KUKA KRL program: MyProgram_344().src

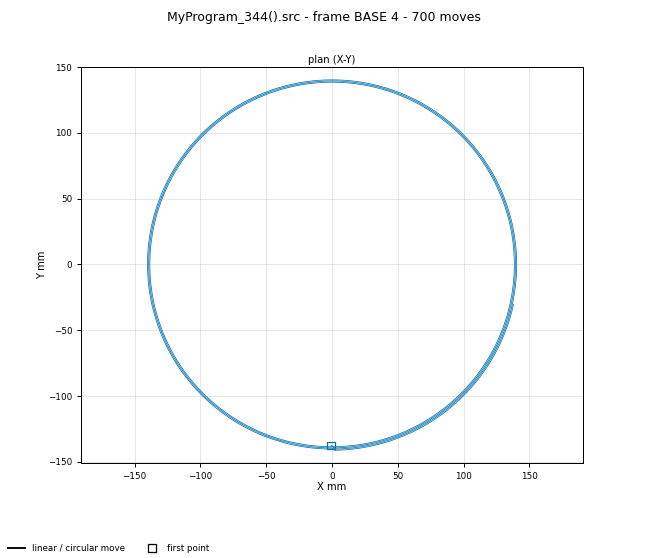
[picture p0: tool path of MyProgram_344().src in frame BASE 4, 700 of 700 moves have a stored position in this frame; points joined in program order, loops and branches not executed]
&ACCESS RVP
&REL 1
&PARAM TEMPLATE = C:\KRC\Roboter\Template\vorgabe
&PARAM EDITMASK = *
DEF MyProgram_344()
; ---- Setting reference (Base) ----
$BASE = BASE_DATA[4]

; --------------------------
; ---- Setting tool (TCP) ----
$TOOL = TOOL_DATA[3]
; --------------------------

$VEL.CP = VEL_APROX_PRINT
Startdeposition()
$VEL.CP = VEL_PRINT
LIN {X -0.555,Y -137.593,Z 192,A -68.2325,B 0.4034,C 0.1604,E1 0.4627,E2 159.7049} C_DIS
Enddeposition()
LIN {X 0.9941,Y -138.4895,Z 192,A -68.6521,B 0.4236,C 0.1629,E1 0.4819,E2 160.302} C_DIS
Startdeposition()
$VEL.CP = VEL_PRINT
LIN {X 0.9941,Y -138.4895,Z 192,A -68.6533,B 0.4236,C 0.1629,E1 0.4819,E2 160.3034} C_DIS
LIN {X -2.5108,Y -138.4702,Z 192,A -70.1889,B 0.423,C 0.1643,E1 0.4773,E2 161.8537} C_DIS
LIN {X -7.0615,Y -138.3127,Z 192,A -71.9031,B 0.4225,C 0.1655,E1 0.4723,E2 163.5419} C_DIS
LIN {X -10.2792,Y -138.1109,Z 192,A -73.1462,B 0.4222,C 0.1664,E1 0.4687,E2 164.7714} C_DIS
LIN {X -14.0249,Y -137.783,Z 192,A -74.535,B 0.4219,C 0.1671,E1 0.4646,E2 166.1344} C_DIS
LIN {X -18.2105,Y -137.2903,Z 192,A -76.1855,B 0.4216,C 0.168,E1 0.4598,E2 167.771} C_DIS
LIN {X -21.5368,Y -136.8082,Z 192,A -77.5051,B 0.4213,C 0.1687,E1 0.4559,E2 169.0801} C_DIS
LIN {X -25.201,Y -136.1828,Z 192,A -78.927,B 0.4211,C 0.1692,E1 0.4518,E2 170.4843} C_DIS
LIN {X -28.0321,Y -135.6266,Z 192,A -80.0916,B 0.4209,C 0.1697,E1 0.4484,E2 171.6448} C_DIS
LIN {X -31.6468,Y -134.8308,Z 192,A -81.5349,B 0.4207,C 0.1701,E1 0.4443,E2 173.0749} C_DIS
LIN {X -34.3072,Y -134.1761,Z 192,A -82.6457,B 0.4206,C 0.1704,E1 0.4411,E2 174.1826} C_DIS
LIN {X -38.108,Y -133.1489,Z 192,A -84.2158,B 0.4205,C 0.1708,E1 0.4366,E2 175.7441} C_DIS
LIN {X -41.3369,Y -132.1821,Z 192,A -85.5836,B 0.4204,C 0.171,E1 0.4327,E2 177.1083} C_DIS
LIN {X -44.1513,Y -131.2668,Z 192,A -86.8094,B 0.4204,C 0.1711,E1 0.4292,E2 178.3348} C_DIS
LIN {X -47.7758,Y -129.9936,Z 192,A -88.3761,B 0.4203,C 0.1711,E1 0.4248,E2 179.8986} C_DIS
LIN {X -50.9793,Y -128.771,Z 192,A -89.8008,B 0.4203,C 0.1711,E1 0.4209,E2 181.325} C_DIS
LIN {X -54.0825,Y -127.4982,Z 192,A -91.2041,B 0.4203,C 0.1711,E1 0.417,E2 182.7313} C_DIS
LIN {X -56.8706,Y -126.2773,Z 192,A -92.5332,B 0.4204,C 0.1709,E1 0.4133,E2 184.0722} C_DIS
LIN {X -60.4865,Y -124.5883,Z 192,A -94.1895,B 0.4206,C 0.1705,E1 0.4089,E2 185.7299} C_DIS
LIN {X -63.61,Y -123.0229,Z 192,A -95.691,B 0.4207,C 0.1701,E1 0.4049,E2 187.2409} C_DIS
LIN {X -66.285,Y -121.6017,Z 192,A -97.0782,B 0.4209,C 0.1697,E1 0.4012,E2 188.65} C_DIS
LIN {X -70.0463,Y -119.4747,Z 192,A -98.9871,B 0.4212,C 0.169,E1 0.3962,E2 190.5788} C_DIS
LIN {X -73.7798,Y -117.2059,Z 192,A -100.9315,B 0.4215,C 0.168,E1 0.3912,E2 192.5456} C_DIS
LIN {X -77.534,Y -114.7569,Z 192,A -102.9321,B 0.422,C 0.1669,E1 0.3862,E2 194.57} C_DIS
LIN {X -81.1785,Y -112.2084,Z 192,A -104.9505,B 0.4225,C 0.1656,E1 0.3813,E2 196.6173} C_DIS
LIN {X -84.7483,Y -109.5372,Z 192,A -106.9996,B 0.4231,C 0.1641,E1 0.3763,E2 198.6993} C_DIS
LIN {X -88.4224,Y -106.5934,Z 192,A -109.1404,B 0.4238,C 0.1623,E1 0.3714,E2 200.871} C_DIS
LIN {X -91.6396,Y -103.8405,Z 192,A -111.1887,B 0.4245,C 0.1605,E1 0.3667,E2 202.9667} C_DIS
LIN {X -94.9496,Y -100.8229,Z 192,A -113.3283,B 0.4253,C 0.1584,E1 0.362,E2 205.1518} C_DIS
LIN {X -98.1617,Y -97.6982,Z 192,A -115.4971,B 0.4261,C 0.156,E1 0.3573,E2 207.3704} C_DIS
LIN {X -101.2932,Y -94.4476,Z 192,A -117.7031,B 0.4271,C 0.1535,E1 0.3527,E2 209.6298} C_DIS
LIN {X -104.4308,Y -90.9664,Z 192,A -119.9695,B 0.4281,C 0.1506,E1 0.3482,E2 211.9476} C_DIS
LIN {X -107.1621,Y -87.7323,Z 192,A -122.1746,B 0.4291,C 0.1477,E1 0.344,E2 214.2236} C_DIS
LIN {X -110.0811,Y -84.0406,Z 192,A -124.5209,B 0.4303,C 0.1443,E1 0.3397,E2 216.6321} C_DIS
LIN {X -112.6171,Y -80.6104,Z 192,A -126.7728,B 0.4314,C 0.1409,E1 0.3357,E2 218.9595} C_DIS
LIN {X -115.2516,Y -76.7967,Z 192,A -129.1574,B 0.4326,C 0.1371,E1 0.3317,E2 221.4161} C_DIS
LIN {X -117.5235,Y -73.2728,Z 192,A -131.4426,B 0.4338,C 0.1333,E1 0.328,E2 223.7857} C_DIS
LIN {X -119.9181,Y -69.2845,Z 192,A -133.8851,B 0.4351,C 0.129,E1 0.3243,E2 226.3071} C_DIS
LIN {X -121.9449,Y -65.6516,Z 192,A -136.1958,B 0.4363,C 0.1248,E1 0.321,E2 228.7072} C_DIS
LIN {X -123.5969,Y -62.4824,Z 192,A -138.0865,B 0.4373,C 0.1211,E1 0.3184,E2 230.6599} C_DIS
LIN {X -125.339,Y -58.9152,Z 192,A -140.2644,B 0.4385,C 0.1168,E1 0.3157,E2 232.9182} C_DIS
LIN {X -126.7762,Y -55.7554,Z 192,A -142.2121,B 0.4395,C 0.1129,E1 0.3133,E2 234.9421} C_DIS
LIN {X -128.1275,Y -52.5756,Z 192,A -144.1677,B 0.4406,C 0.1088,E1 0.3111,E2 236.9756} C_DIS
LIN {X -129.393,Y -49.3792,Z 192,A -146.1301,B 0.4416,C 0.1047,E1 0.309,E2 239.0175} C_DIS
LIN {X -130.5727,Y -46.1694,Z 192,A -148.0979,B 0.4426,C 0.1004,E1 0.307,E2 241.0662} C_DIS
LIN {X -131.4708,Y -43.5386,Z 192,A -149.7078,B 0.4434,C 0.0968,E1 0.3055,E2 242.7429} C_DIS
LIN {X -132.529,Y -40.2034,Z 192,A -151.7407,B 0.4443,C 0.0922,E1 0.3037,E2 244.8603} C_DIS
LIN {X -133.4355,Y -37.0832,Z 192,A -153.656,B 0.4452,C 0.0878,E1 0.3022,E2 246.8574} C_DIS
LIN {X -134.2916,Y -33.8522,Z 192,A -155.631,B 0.4461,C 0.0832,E1 0.3007,E2 248.9165} C_DIS
LIN {X -135.1229,Y -30.3677,Z 192,A -157.7323,B 0.447,C 0.0782,E1 0.2993,E2 251.1051} C_DIS
LIN {X -135.8753,Y -26.8097,Z 192,A -159.9357,B 0.4479,C 0.0729,E1 0.298,E2 253.4062} C_DIS
LIN {X -136.6401,Y -22.5773,Z 192,A -162.5203,B 0.4489,C 0.0665,E1 0.2967,E2 256.102} C_DIS
LIN {X -137.1281,Y -19.3939,Z 192,A -164.4714,B 0.4496,C 0.0617,E1 0.2959,E2 258.1376} C_DIS
LIN {X -137.6124,Y -15.6101,Z 192,A -166.7803,B 0.4504,C 0.0559,E1 0.2951,E2 260.5455} C_DIS
LIN {X -138.0192,Y -11.4448,Z 192,A -169.4132,B 0.4511,C 0.0493,E1 0.2943,E2 263.2988} C_DIS
LIN {X -138.3076,Y -7.1633,Z 192,A -172.0124,B 0.4518,C 0.0427,E1 0.2939,E2 266.0064} C_DIS
LIN {X -138.4451,Y -3.6396,Z 192,A -174.1874,B 0.4523,C 0.0371,E1 0.2937,E2 268.2745} C_DIS
LIN {X -138.4943,Y -0.3953,Z 192,A -176.1959,B 0.4527,C 0.0319,E1 0.2937,E2 270.3685} C_DIS
LIN {X -138.4702,Y 2.5108,Z 192,A -177.963,B 0.453,C 0.0274,E1 0.2937,E2 272.2073} C_DIS
LIN {X -138.3076,Y 7.1633,Z 192,A 179.1755,B 0.4534,C 0.02,E1 0.2941,E2 275.1859} C_DIS
LIN {X -138.3076,Y 7.1633,Z 192,A 179.1746,B 0.4534,C 0.02,E1 0.2941,E2 275.1869} C_DIS
LIN {X -137.9693,Y 12.0354,Z 192,A 176.2175,B 0.4536,C 0.0124,E1 0.2947,E2 278.2592} C_DIS
LIN {X -137.9693,Y 12.0354,Z 192,A 176.2165,B 0.4536,C 0.0124,E1 0.2947,E2 278.2602} C_DIS
LIN {X -137.6124,Y 15.6101,Z 192,A 174.0658,B 0.4538,C 0.0069,E1 0.2954,E2 280.4913} C_DIS
LIN {X -137.214,Y 18.7931,Z 192,A 172.1065,B 0.4538,C 0.0019,E1 0.2961,E2 282.5262} C_DIS
LIN {X -136.7379,Y 21.9909,Z 192,A 170.138,B 0.4538,C -0.0031,E1 0.297,E2 284.569} C_DIS
LIN {X -136.2264,Y 24.9574,Z 192,A 168.3314,B 0.4538,C -0.0076,E1 0.2979,E2 286.4408} C_DIS
LIN {X -135.5475,Y 28.4205,Z 192,A 166.1798,B 0.4536,C -0.013,E1 0.2991,E2 288.6719} C_DIS
LIN {X -134.8308,Y 31.6468,Z 192,A 164.192,B 0.4535,C -0.0179,E1 0.3004,E2 290.7298} C_DIS
LIN {X -134.0315,Y 34.877,Z 192,A 162.2011,B 0.4532,C -0.0227,E1 0.3018,E2 292.7892} C_DIS
LIN {X -133.2966,Y 37.5799,Z 192,A 160.5251,B 0.453,C -0.0267,E1 0.3031,E2 294.522} C_DIS
LIN {X -132.1821,Y 41.3369,Z 192,A 158.2172,B 0.4527,C -0.0322,E1 0.3051,E2 296.9044} C_DIS
LIN {X -131.1305,Y 44.5606,Z 192,A 156.2264,B 0.4523,C -0.0368,E1 0.3069,E2 298.9579} C_DIS
LIN {X -130.0987,Y 47.4843,Z 192,A 154.4441,B 0.452,C -0.0409,E1 0.3087,E2 300.7927} C_DIS
LIN {X -128.9199,Y 50.5962,Z 192,A 152.4488,B 0.4515,C -0.0453,E1 0.3108,E2 302.8522} C_DIS
LIN {X -127.4626,Y 54.1678,Z 192,A 150.2777,B 0.451,C -0.0501,E1 0.3132,E2 305.082} C_DIS
LIN {X -126.0683,Y 57.338,Z 192,A 148.3077,B 0.4505,C -0.0543,E1 0.3156,E2 307.106} C_DIS
LIN {X -124.5883,Y 60.4865,Z 192,A 146.3461,B 0.45,C -0.0584,E1 0.3181,E2 309.1192} C_DIS
LIN {X -123.0229,Y 63.61,Z 192,A 144.3948,B 0.4495,C -0.0624,E1 0.3207,E2 311.1199} C_DIS
LIN {X -121.5263,Y 66.4232,Z 192,A 142.5706,B 0.449,C -0.066,E1 0.3232,E2 312.9928} C_DIS
LIN {X -119.4747,Y 70.0463,Z 192,A 140.2278,B 0.4483,C -0.0704,E1 0.3267,E2 315.3943} C_DIS
LIN {X -117.1798,Y 73.8211,Z 192,A 137.8387,B 0.4476,C -0.0748,E1 0.3304,E2 317.8354} C_DIS
LIN {X -114.7569,Y 77.534,Z 192,A 135.4725,B 0.4469,C -0.0789,E1 0.3343,E2 320.2501} C_DIS
LIN {X -112.2084,Y 81.1785,Z 192,A 133.1307,B 0.4462,C -0.0828,E1 0.3383,E2 322.6369} C_DIS
LIN {X -109.5372,Y 84.7483,Z 192,A 130.8146,B 0.4455,C -0.0865,E1 0.3424,E2 324.9946} C_DIS
LIN {X -106.5934,Y 88.4224,Z 192,A 128.4626,B 0.4448,C -0.09,E1 0.3468,E2 327.3815} C_DIS
LIN {X -103.8405,Y 91.6396,Z 192,A 126.265,B 0.4442,C -0.0931,E1 0.3511,E2 329.6173} C_DIS
LIN {X -100.8229,Y 94.9496,Z 192,A 124.0464,B 0.4435,C -0.096,E1 0.3556,E2 331.8666} C_DIS
LIN {X -97.6982,Y 98.1617,Z 192,A 121.8322,B 0.4429,C -0.0987,E1 0.3603,E2 334.1107} C_DIS
LIN {X -94.2952,Y 101.4351,Z 192,A 119.6016,B 0.4424,C -0.1012,E1 0.3651,E2 336.3638} C_DIS
LIN {X -90.9664,Y 104.4308,Z 192,A 117.4631,B 0.4419,C -0.1034,E1 0.3699,E2 338.5252} C_DIS
LIN {X -87.7323,Y 107.1621,Z 192,A 115.4142,B 0.4414,C -0.1053,E1 0.3746,E2 340.598} C_DIS
LIN {X -84.0406,Y 110.0811,Z 192,A 113.2812,B 0.441,C -0.1072,E1 0.3796,E2 342.7453} C_DIS
LIN {X -80.4554,Y 112.728,Z 192,A 111.2383,B 0.4406,C -0.1087,E1 0.3845,E2 344.8035} C_DIS
LIN {X -76.9626,Y 115.1409,Z 192,A 109.2749,B 0.4403,C -0.11,E1 0.3894,E2 346.783} C_DIS
LIN {X -73.2728,Y 117.5235,Z 192,A 107.304,B 0.44,C -0.1111,E1 0.3944,E2 348.7653} C_DIS
LIN {X -69.2845,Y 119.9181,Z 192,A 105.3033,B 0.4397,C -0.1121,E1 0.3995,E2 350.7712} C_DIS
LIN {X -65.7176,Y 121.9094,Z 192,A 103.4573,B 0.4396,C -0.1128,E1 0.4044,E2 352.629} C_DIS
LIN {X -62.0516,Y 123.8162,Z 192,A 101.7909,B 0.4394,C -0.1134,E1 0.4088,E2 354.2911} C_DIS
LIN {X -59.3101,Y 125.1503,Z 192,A 100.4556,B 0.4394,C -0.1137,E1 0.4124,E2 355.6316} C_DIS
LIN {X -55.7554,Y 126.7762,Z 192,A 98.838,B 0.4393,C -0.114,E1 0.4168,E2 357.2487} C_DIS
LIN {X -52.5756,Y 128.1275,Z 192,A 97.3919,B 0.4393,C -0.1141,E1 0.4208,E2 358.6955} C_DIS
LIN {X -49.6556,Y 129.2856,Z 192,A 96.0714,B 0.4393,C -0.1141,E1 0.4245,E2 360.017} C_DIS
LIN {X -46.1694,Y 130.5727,Z 192,A 94.5588,B 0.4393,C -0.1141,E1 0.4287,E2 361.527} C_DIS
LIN {X -42.9496,Y 131.667,Z 192,A 93.172,B 0.4393,C -0.114,E1 0.4326,E2 362.9116} C_DIS
LIN {X -39.967,Y 132.6014,Z 192,A 91.8954,B 0.4393,C -0.1137,E1 0.4362,E2 364.1863} C_DIS
LIN {X -36.4926,Y 133.6007,Z 192,A 90.4567,B 0.4394,C -0.1134,E1 0.4404,E2 365.6199} C_DIS
LIN {X -33.2616,Y 134.4415,Z 192,A 89.1274,B 0.4395,C -0.1131,E1 0.4442,E2 366.9444} C_DIS
LIN {X -30.033,Y 135.1994,Z 192,A 87.817,B 0.4396,C -0.1126,E1 0.448,E2 368.2492} C_DIS
LIN {X -27.3611,Y 135.7631,Z 192,A 86.6941,B 0.4397,C -0.1121,E1 0.4513,E2 369.3711} C_DIS
LIN {X -23.5946,Y 136.4703,Z 192,A 85.2526,B 0.4399,C -0.1115,E1 0.4554,E2 370.8004} C_DIS
LIN {X -20.3903,Y 136.9857,Z 192,A 83.9977,B 0.4401,C -0.1108,E1 0.4591,E2 372.0478} C_DIS
LIN {X -17.1996,Y 137.4228,Z 192,A 82.7606,B 0.4402,C -0.1101,E1 0.4627,E2 373.2766} C_DIS
LIN {X -13.0223,Y 137.8793,Z 192,A 81.1595,B 0.4405,C -0.1091,E1 0.4674,E2 374.8657} C_DIS
LIN {X -9.967,Y 138.1337,Z 192,A 79.9863,B 0.4407,C -0.1083,E1 0.4709,E2 376.0306} C_DIS
LIN {X -6.1741,Y 138.3573,Z 192,A 78.5706,B 0.441,C -0.1072,E1 0.475,E2 377.4331} C_DIS
LIN {X -3.6396,Y 138.4451,Z 192,A 77.5718,B 0.4412,C -0.1063,E1 0.478,E2 378.4273} C_DIS
LIN {X 0,Y 138.495,Z 192,A 76.2697,B 0.4414,C -0.1053,E1 0.4818,E2 379.712} C_DIS
LIN {X 4.1288,Y 138.4315,Z 192,A 74.7561,B 0.4418,C -0.1039,E1 0.4862,E2 381.2087} C_DIS
LIN {X 7.1633,Y 138.3076,Z 192,A 73.5697,B 0.442,C -0.1027,E1 0.4897,E2 382.3889} C_DIS
LIN {X 10.8687,Y 138.0678,Z 192,A 72.2626,B 0.4423,C -0.1014,E1 0.4935,E2 383.6763} C_DIS
LIN {X 14.0249,Y 137.783,Z 192,A 71.1092,B 0.4426,C -0.1001,E1 0.4968,E2 384.8159} C_DIS
LIN {X 18.3405,Y 137.2733,Z 192,A 69.5037,B 0.443,C -0.0983,E1 0.5015,E2 386.4043} C_DIS
LIN {X 21.9321,Y 136.747,Z 192,A 68.2316,B 0.4434,C -0.0968,E1 0.5051,E2 387.6564} C_DIS
LIN {X 24.721,Y 136.2687,Z 192,A 67.1837,B 0.4436,C -0.0955,E1 0.5081,E2 388.6932} C_DIS
LIN {X 28.4205,Y 135.5475,Z 192,A 65.879,B 0.444,C -0.0939,E1 0.5118,E2 389.9755} C_DIS
LIN {X 32.7749,Y 134.5588,Z 192,A 64.2612,B 0.4445,C -0.0917,E1 0.5164,E2 391.5725} C_DIS
LIN {X 36.4926,Y 133.6007,Z 192,A 62.9482,B 0.4448,C -0.0899,E1 0.52,E2 392.8609} C_DIS
LIN {X 39.7229,Y 132.6761,Z 192,A 61.7715,B 0.4451,C -0.0882,E1 0.5233,E2 394.0183} C_DIS
LIN {X 42.5024,Y 131.8098,Z 192,A 60.724,B 0.4455,C -0.0867,E1 0.5261,E2 395.0513} C_DIS
LIN {X 46.1694,Y 130.5727,Z 192,A 59.4127,B 0.4458,C -0.0847,E1 0.5297,E2 396.3362} C_DIS
LIN {X 49.3792,Y 129.393,Z 192,A 58.2311,B 0.4462,C -0.0829,E1 0.5328,E2 397.4964} C_DIS
LIN {X 52.0629,Y 128.3342,Z 192,A 57.2312,B 0.4465,C -0.0813,E1 0.5355,E2 398.4782} C_DIS
LIN {X 55.7554,Y 126.7762,Z 192,A 55.8629,B 0.4469,C -0.0791,E1 0.5391,E2 399.8196} C_DIS
LIN {X 58.4713,Y 125.5442,Z 192,A 54.811,B 0.4472,C -0.0773,E1 0.5418,E2 400.8542} C_DIS
LIN {X 62.7685,Y 123.4512,Z 192,A 53.2475,B 0.4476,C -0.0747,E1 0.5458,E2 402.3785} C_DIS
LIN {X 65.9341,Y 121.7931,Z 192,A 51.9114,B 0.448,C -0.0723,E1 0.5491,E2 403.7011} C_DIS
LIN {X 69.7683,Y 119.638,Z 192,A 50.4277,B 0.4484,C -0.0696,E1 0.5528,E2 405.1525} C_DIS
LIN {X 73.5368,Y 117.3592,Z 192,A 48.9472,B 0.4488,C -0.0669,E1 0.5563,E2 406.6} C_DIS
LIN {X 77.2651,Y 114.939,Z 192,A 47.4954,B 0.4492,C -0.0643,E1 0.5597,E2 408.0139} C_DIS
LIN {X 80.9148,Y 112.3995,Z 192,A 46.0136,B 0.4496,C -0.0615,E1 0.5631,E2 409.4604} C_DIS
LIN {X 84.4903,Y 109.7372,Z 192,A 44.4994,B 0.45,C -0.0585,E1 0.5665,E2 410.9417} C_DIS
LIN {X 87.9854,Y 106.9552,Z 192,A 43.0481,B 0.4504,C -0.0556,E1 0.5696,E2 412.3531} C_DIS
LIN {X 91.3943,Y 104.0574,Z 192,A 41.5465,B 0.4508,C -0.0526,E1 0.5728,E2 413.8193} C_DIS
LIN {X 94.7112,Y 101.0477,Z 192,A 40.0745,B 0.4511,C -0.0496,E1 0.5758,E2 415.2523} C_DIS
LIN {X 97.9307,Y 97.9307,Z 192,A 38.6398,B 0.4514,C -0.0467,E1 0.5786,E2 416.6436} C_DIS
LIN {X 101.0477,Y 94.7112,Z 192,A 37.1759,B 0.4517,C -0.0436,E1 0.5814,E2 418.0669} C_DIS
LIN {X 103.9957,Y 91.4641,Z 192,A 35.739,B 0.452,C -0.0405,E1 0.5841,E2 419.464} C_DIS
LIN {X 106.9552,Y 87.9854,Z 192,A 34.2626,B 0.4523,C -0.0374,E1 0.5867,E2 420.8964} C_DIS
LIN {X 109.7372,Y 84.4903,Z 192,A 32.8039,B 0.4525,C -0.0342,E1 0.5891,E2 422.3133} C_DIS
LIN {X 112.3995,Y 80.9148,Z 192,A 31.3402,B 0.4528,C -0.0309,E1 0.5915,E2 423.7358} C_DIS
LIN {X 114.939,Y 77.2651,Z 192,A 29.9377,B 0.453,C -0.0279,E1 0.5937,E2 425.0905} C_DIS
LIN {X 117.352,Y 73.5484,Z 192,A 28.5103,B 0.4531,C -0.0247,E1 0.5958,E2 426.4731} C_DIS
LIN {X 119.638,Y 69.7683,Z 192,A 27.0552,B 0.4533,C -0.0213,E1 0.5978,E2 427.8868} C_DIS
LIN {X 121.875,Y 65.7816,Z 192,A 25.6074,B 0.4535,C -0.0181,E1 0.5997,E2 429.2848} C_DIS
LIN {X 123.8162,Y 62.0516,Z 192,A 24.332,B 0.4535,C -0.0152,E1 0.6013,E2 430.5074} C_DIS
LIN {X 125.339,Y 58.9152,Z 192,A 23.2157,B 0.4536,C -0.0127,E1 0.6026,E2 431.5864} C_DIS
LIN {X 126.7762,Y 55.7554,Z 192,A 22.1058,B 0.4536,C -0.0101,E1 0.6038,E2 432.6588} C_DIS
LIN {X 127.9883,Y 52.9089,Z 192,A 21.1185,B 0.4537,C -0.0078,E1 0.6049,E2 433.6121} C_DIS
LIN {X 129.393,Y 49.3792,Z 192,A 19.9048,B 0.4537,C -0.005,E1 0.6061,E2 434.784} C_DIS
LIN {X 130.361,Y 46.7567,Z 192,A 19.0109,B 0.4538,C -0.0029,E1 0.6069,E2 435.647} C_DIS
LIN {X 131.5332,Y 43.3512,Z 192,A 17.8438,B 0.4538,C -0.0001,E1 0.6079,E2 436.776} C_DIS
LIN {X 132.6761,Y 39.7229,Z 192,A 16.6541,B 0.4538,C 0.0026,E1 0.6088,E2 437.92} C_DIS
LIN {X 133.8705,Y 35.4808,Z 192,A 15.2396,B 0.4538,C 0.006,E1 0.6098,E2 439.2855} C_DIS
LIN {X 134.8308,Y 31.6468,Z 192,A 13.9948,B 0.4538,C 0.0089,E1 0.6106,E2 440.4832} C_DIS
LIN {X 135.5475,Y 28.4205,Z 192,A 12.9443,B 0.4537,C 0.0114,E1 0.6112,E2 441.4951} C_DIS
LIN {X 136.1828,Y 25.201,Z 192,A 11.9014,B 0.4536,C 0.0139,E1 0.6118,E2 442.4996} C_DIS
LIN {X 136.8951,Y 20.9756,Z 192,A 10.5272,B 0.4535,C 0.0172,E1 0.6124,E2 443.8247} C_DIS
LIN {X 137.4228,Y 17.1996,Z 192,A 9.3297,B 0.4534,C 0.02,E1 0.6128,E2 444.9751} C_DIS
LIN {X 137.8793,Y 13.0223,Z 192,A 7.9962,B 0.4532,C 0.0232,E1 0.6132,E2 446.258} C_DIS
LIN {X 138.1406,Y 9.8725,Z 192,A 6.9929,B 0.4531,C 0.0256,E1 0.6134,E2 447.223} C_DIS
LIN {X 138.3357,Y 6.6024,Z 192,A 5.959,B 0.4529,C 0.028,E1 0.6135,E2 448.2163} C_DIS
LIN {X 138.4451,Y 3.6396,Z 192,A 4.9707,B 0.4528,C 0.0304,E1 0.6136,E2 449.1745} C_DIS
LIN {X 138.4943,Y 0.3953,Z 192,A 3.9518,B 0.4526,C 0.0328,E1 0.6136,E2 450.1521} C_DIS
LIN {X 138.4608,Y -3.074,Z 192,A 2.875,B 0.4524,C 0.0353,E1 0.6136,E2 451.1829} C_DIS
LIN {X 138.3076,Y -7.1633,Z 192,A 1.5785,B 0.4522,C 0.0384,E1 0.6134,E2 452.4282} C_DIS
LIN {X 138.087,Y -10.6067,Z 192,A 0.4731,B 0.452,C 0.041,E1 0.6132,E2 453.4917} C_DIS
LIN {X 137.783,Y -14.0249,Z 192,A -0.625,B 0.4517,C 0.0436,E1 0.6129,E2 454.548} C_DIS
LIN {X 137.4921,Y -16.6185,Z 192,A -1.5008,B 0.4515,C 0.0458,E1 0.6127,E2 455.3971} C_DIS
LIN {X 136.9857,Y -20.3903,Z 192,A -2.673,B 0.4512,C 0.0484,E1 0.6122,E2 456.5163} C_DIS
LIN {X 136.4839,Y -23.5132,Z 192,A -3.6749,B 0.451,C 0.0508,E1 0.6118,E2 457.4775} C_DIS
LIN {X 135.8753,Y -26.8097,Z 192,A -4.7551,B 0.4507,C 0.0533,E1 0.6113,E2 458.517} C_DIS
LIN {X 135.1994,Y -30.033,Z 192,A -5.8083,B 0.4504,C 0.0558,E1 0.6107,E2 459.5289} C_DIS
LIN {X 134.4416,Y -33.2616,Z 192,A -6.8713,B 0.4501,C 0.0582,E1 0.61,E2 460.5505} C_DIS
LIN {X 133.7106,Y -36.0806,Z 192,A -7.826,B 0.4498,C 0.0605,E1 0.6093,E2 461.4714} C_DIS
LIN {X 132.6761,Y -39.7229,Z 192,A -9.016,B 0.4494,C 0.0632,E1 0.6084,E2 462.6105} C_DIS
LIN {X 131.667,Y -42.9496,Z 192,A -10.1007,B 0.449,C 0.0656,E1 0.6075,E2 463.6524} C_DIS
LIN {X 130.5727,Y -46.1694,Z 192,A -11.1926,B 0.4487,C 0.0681,E1 0.6066,E2 464.7013} C_DIS
LIN {X 129.59,Y -48.8533,Z 192,A -12.1224,B 0.4483,C 0.0702,E1 0.6057,E2 465.5964} C_DIS
LIN {X 128.1275,Y -52.5756,Z 192,A -13.3979,B 0.4479,C 0.0731,E1 0.6044,E2 466.8197} C_DIS
LIN {X 126.7762,Y -55.7554,Z 192,A -14.5111,B 0.4475,C 0.0756,E1 0.6032,E2 467.8892} C_DIS
LIN {X 125.339,Y -58.9152,Z 192,A -15.6306,B 0.447,C 0.0781,E1 0.602,E2 468.9647} C_DIS
LIN {X 123.8968,Y -61.8883,Z 192,A -16.693,B 0.4466,C 0.0804,E1 0.6007,E2 469.9845} C_DIS
LIN {X 122.3814,Y -64.8316,Z 192,A -17.7503,B 0.4462,C 0.0827,E1 0.5994,E2 470.9981} C_DIS
LIN {X 120.5157,Y -68.2408,Z 192,A -19.0826,B 0.4456,C 0.0857,E1 0.5976,E2 472.2919} C_DIS
LIN {X 118.2823,Y -72.0428,Z 192,A -20.5134,B 0.445,C 0.0888,E1 0.5956,E2 473.6671} C_DIS
LIN {X 115.9812,Y -75.691,Z 192,A -21.9254,B 0.4444,C 0.0918,E1 0.5936,E2 475.0263} C_DIS
LIN {X 113.4302,Y -79.4635,Z 192,A -23.3998,B 0.4438,C 0.0949,E1 0.5913,E2 476.4424} C_DIS
LIN {X 110.8167,Y -83.0694,Z 192,A -24.8543,B 0.4431,C 0.0979,E1 0.5889,E2 477.8414} C_DIS
LIN {X 108.101,Y -86.5737,Z 192,A -26.327,B 0.4424,C 0.1009,E1 0.5865,E2 479.2621} C_DIS
LIN {X 105.2302,Y -90.0415,Z 192,A -27.7831,B 0.4418,C 0.1038,E1 0.5839,E2 480.6596} C_DIS
LIN {X 102.2647,Y -93.3958,Z 192,A -29.2565,B 0.4411,C 0.1067,E1 0.5812,E2 482.078} C_DIS
LIN {X 99.2163,Y -96.6279,Z 192,A -30.7254,B 0.4404,C 0.1096,E1 0.5784,E2 483.4932} C_DIS
LIN {X 96.011,Y -99.8135,Z 192,A -32.2504,B 0.4396,C 0.1126,E1 0.5754,E2 484.9679} C_DIS
LIN {X 92.7324,Y -102.8667,Z 192,A -33.7377,B 0.4389,C 0.1154,E1 0.5724,E2 486.4016} C_DIS
LIN {X 89.5033,Y -105.6877,Z 192,A -35.0973,B 0.4383,C 0.1178,E1 0.5696,E2 487.6999} C_DIS
LIN {X 86.1302,Y -108.454,Z 192,A -36.5622,B 0.4375,C 0.1205,E1 0.5664,E2 489.1147} C_DIS
LIN {X 82.6157,Y -111.1545,Z 192,A -38.052,B 0.4368,C 0.1231,E1 0.5632,E2 490.5535} C_DIS
LIN {X 79.0004,Y -113.7524,Z 192,A -39.5497,B 0.436,C 0.1258,E1 0.5598,E2 492.0001} C_DIS
LIN {X 75.5139,Y -116.0962,Z 192,A -41.0032,B 0.4353,C 0.1283,E1 0.5564,E2 493.4114} C_DIS
LIN {X 71.7664,Y -118.4494,Z 192,A -42.5021,B 0.4346,C 0.1308,E1 0.5528,E2 494.8607} C_DIS
LIN {X 67.9604,Y -120.6733,Z 192,A -44.0032,B 0.4338,C 0.1332,E1 0.5492,E2 496.3135} C_DIS
LIN {X 64.0989,Y -122.7662,Z 192,A -45.4473,B 0.4331,C 0.1354,E1 0.5457,E2 497.7011} C_DIS
LIN {X 60.4865,Y -124.5883,Z 192,A -46.8242,B 0.4325,C 0.1375,E1 0.5422,E2 499.0334} C_DIS
LIN {X 57.7806,Y -125.8636,Z 192,A -47.8847,B 0.4319,C 0.1392,E1 0.5395,E2 500.0672} C_DIS
LIN {X 54.1678,Y -127.4626,Z 192,A -49.2201,B 0.4313,C 0.1411,E1 0.536,E2 501.3574} C_DIS
LIN {X 50.9793,Y -128.771,Z 192,A -50.4163,B 0.4308,C 0.1428,E1 0.5329,E2 502.5188} C_DIS
LIN {X 48.0728,Y -129.8823,Z 192,A -51.5145,B 0.4302,C 0.1444,E1 0.53,E2 503.5883} C_DIS
LIN {X 44.5606,Y -131.1305,Z 192,A -52.8035,B 0.4297,C 0.1461,E1 0.5266,E2 504.8388} C_DIS
LIN {X 41.9266,Y -131.9938,Z 192,A -53.7841,B 0.4292,C 0.1474,E1 0.5239,E2 505.7942} C_DIS
LIN {X 38.6732,Y -132.9834,Z 192,A -54.9796,B 0.4287,C 0.1489,E1 0.5207,E2 506.9575} C_DIS
LIN {X 34.877,Y -134.0315,Z 192,A -56.3689,B 0.4281,C 0.1507,E1 0.5168,E2 508.3102} C_DIS
LIN {X 31.6468,Y -134.8308,Z 192,A -57.5522,B 0.4276,C 0.1521,E1 0.5135,E2 509.4641} C_DIS
LIN {X 28.4205,Y -135.5475,Z 192,A -58.7326,B 0.4271,C 0.1535,E1 0.5102,E2 510.6159} C_DIS
LIN {X 25.201,Y -136.1828,Z 192,A -59.9103,B 0.4266,C 0.1548,E1 0.5069,E2 511.7661} C_DIS
LIN {X 22.4273,Y -136.6651,Z 192,A -60.953,B 0.4262,C 0.156,E1 0.504,E2 512.7903} C_DIS
LIN {X 18.7931,Y -137.214,Z 192,A -62.2549,B 0.4257,C 0.1573,E1 0.5003,E2 514.0586} C_DIS
LIN {X 15.6101,Y -137.6124,Z 192,A -63.4217,B 0.4252,C 0.1585,E1 0.4969,E2 515.2009} C_DIS
LIN {X 11.4448,Y -138.0192,Z 192,A -64.9524,B 0.4247,C 0.1599,E1 0.4925,E2 516.7008} C_DIS
LIN {X 8.3309,Y -138.2421,Z 192,A -66.1418,B 0.4243,C 0.1611,E1 0.4891,E2 517.8748} C_DIS
LIN {X 4.6209,Y -138.4179,Z 192,A -67.4751,B 0.4239,C 0.1621,E1 0.4852,E2 519.1767} C_DIS
LIN {X 1.5336,Y -138.4865,Z 192,A -68.6233,B 0.4235,C 0.1631,E1 0.4819,E2 520.3051} C_DIS
LIN {X 1.5336,Y -138.4865,Z 192,A -68.6233,B 0.4235,C 0.1631,E1 0.4819,E2 520.3051} C_DIS
Enddeposition()
LIN {X 1.0026,Y -139.3847,Z 192,A -69.1006,B 0.4435,C 0.1645,E1 0.5006,E2 520.8324} C_DIS
Startdeposition()
$VEL.CP = VEL_PRINT
LIN {X 4.2647,Y -139.327,Z 192,A -67.6877,B 0.444,C 0.1631,E1 0.5048,E2 519.4071} C_DIS
LIN {X 8.4179,Y -139.1373,Z 192,A -66.1532,B 0.4445,C 0.1618,E1 0.5092,E2 517.8995} C_DIS
LIN {X 12.2098,Y -138.8567,Z 192,A -64.8025,B 0.4449,C 0.1606,E1 0.5131,E2 516.5817} C_DIS
LIN {X 15.533,Y -138.5248,Z 192,A -63.5851,B 0.4453,C 0.1595,E1 0.5166,E2 515.3884} C_DIS
LIN {X 18.4825,Y -138.1613,Z 192,A -62.4978,B 0.4457,C 0.1584,E1 0.5197,E2 514.3216} C_DIS
LIN {X 22.1548,Y -137.6219,Z 192,A -61.0215,B 0.4463,C 0.1566,E1 0.5239,E2 512.8521} C_DIS
LIN {X 29.1089,Y -136.3185,Z 192,A -58.742,B 0.447,C 0.1546,E1 0.5302,E2 510.671} C_DIS
LIN {X 33.2706,Y -135.364,Z 192,A -57.0664,B 0.4478,C 0.1523,E1 0.5349,E2 509.0067} C_DIS
LIN {X 35.8565,Y -134.7007,Z 192,A -56.0558,B 0.4482,C 0.151,E1 0.5378,E2 508.009} C_DIS
LIN {X 39.3465,Y -133.723,Z 192,A -54.798,B 0.4488,C 0.1495,E1 0.5412,E2 506.7871} C_DIS
LIN {X 43.33,Y -132.4877,Z 192,A -53.3837,B 0.4493,C 0.1477,E1 0.545,E2 505.4191} C_DIS
LIN {X 45.9063,Y -131.6154,Z 192,A -52.3661,B 0.4498,C 0.1462,E1 0.5477,E2 504.4164} C_DIS
LIN {X 49.3442,Y -130.366,Z 192,A -51.1206,B 0.4504,C 0.1446,E1 0.551,E2 503.2106} C_DIS
LIN {X 52.5632,Y -129.1017,Z 192,A -49.8788,B 0.4509,C 0.1428,E1 0.5543,E2 501.996} C_DIS
LIN {X 56.147,Y -127.5857,Z 192,A -48.2348,B 0.4519,C 0.1398,E1 0.5587,E2 500.3437} C_DIS
LIN {X 59.6467,Y -125.9857,Z 192,A -47.3378,B 0.452,C 0.1393,E1 0.5607,E2 499.5532} C_DIS
LIN {X 62.4051,Y -124.6442,Z 192,A -46.1726,B 0.4526,C 0.1373,E1 0.5637,E2 498.402} C_DIS
LIN {X 65.3981,Y -123.0993,Z 192,A -45.016,B 0.4532,C 0.1355,E1 0.5666,E2 497.28} C_DIS
LIN {X 69.6684,Y -120.7345,Z 192,A -43.2878,B 0.454,C 0.1326,E1 0.5708,E2 495.5937} C_DIS
LIN {X 73.349,Y -118.5348,Z 192,A -41.8003,B 0.4548,C 0.1301,E1 0.5744,E2 494.1476} C_DIS
LIN {X 77.1511,Y -116.0959,Z 192,A -40.2722,B 0.4555,C 0.1275,E1 0.5779,E2 492.669} C_DIS
LIN {X 80.8132,Y -113.5773,Z 192,A -38.7551,B 0.4562,C 0.1249,E1 0.5814,E2 491.1984} C_DIS
LIN {X 84.4876,Y -110.8709,Z 192,A -37.2394,B 0.4569,C 0.1222,E1 0.5847,E2 489.7368} C_DIS
LIN {X 87.9766,Y -108.1234,Z 192,A -35.7468,B 0.4576,C 0.1195,E1 0.5879,E2 488.294} C_DIS
LIN {X 91.3702,Y -105.2714,Z 192,A -34.2501,B 0.4584,C 0.1168,E1 0.5911,E2 486.8457} C_DIS
LIN {X 94.8453,Y -102.1512,Z 192,A -32.7127,B 0.4591,C 0.1139,E1 0.5942,E2 485.3652} C_DIS
LIN {X 98.0714,Y -99.0582,Z 192,A -31.2421,B 0.4598,C 0.1111,E1 0.5971,E2 483.9488} C_DIS
LIN {X 101.1735,Y -95.8878,Z 192,A -29.7481,B 0.4605,C 0.1082,E1 0.5999,E2 482.5033} C_DIS
LIN {X 104.2757,Y -92.5046,Z 192,A -28.2613,B 0.4611,C 0.1053,E1 0.6026,E2 481.0754} C_DIS
LIN {X 107.1472,Y -89.163,Z 192,A -26.7883,B 0.4618,C 0.1023,E1 0.6052,E2 479.6518} C_DIS
LIN {X 109.995,Y -85.625,Z 192,A -25.3246,B 0.4624,C 0.0994,E1 0.6077,E2 478.247} C_DIS
LIN {X 112.5674,Y -82.2142,Z 192,A -23.9253,B 0.4631,C 0.0965,E1 0.61,E2 476.8995} C_DIS
LIN {X 115.0601,Y -78.6872,Z 192,A -22.5102,B 0.4637,C 0.0935,E1 0.6122,E2 475.5364} C_DIS
LIN {X 117.6047,Y -74.8315,Z 192,A -20.6367,B 0.4646,C 0.0888,E1 0.615,E2 473.6653} C_DIS
LIN {X 120.1464,Y -70.6775,Z 192,A -19.6955,B 0.4647,C 0.0881,E1 0.6162,E2 472.8786} C_DIS
LIN {X 120.1464,Y -70.6775,Z 192,A -19.6964,B 0.4647,C 0.0881,E1 0.6162,E2 472.8797} C_DIS
LIN {X 122.5672,Y -66.3921,Z 192,A -17.7973,B 0.4656,C 0.0834,E1 0.6187,E2 470.9972} C_DIS
LIN {X 124.383,Y -62.9196,Z 192,A -16.6332,B 0.466,C 0.0811,E1 0.6201,E2 469.8967} C_DIS
LIN {X 126.5614,Y -58.4133,Z 192,A -14.9731,B 0.4666,C 0.0773,E1 0.6221,E2 468.2926} C_DIS
LIN {X 128.3062,Y -54.4805,Z 192,A -13.6205,B 0.4671,C 0.0744,E1 0.6235,E2 466.9986} C_DIS
LIN {X 129.3571,Y -51.9297,Z 192,A -12.7257,B 0.4674,C 0.0724,E1 0.6244,E2 466.1372} C_DIS
LIN {X 130.6249,Y -48.6532,Z 192,A -11.5589,B 0.4678,C 0.0697,E1 0.6256,E2 465.0088} C_DIS
LIN {X 132.0167,Y -44.7445,Z 192,A -10.287,B 0.4682,C 0.0669,E1 0.6267,E2 463.7974} C_DIS
LIN {X 133.4569,Y -40.2433,Z 192,A -8.6937,B 0.4688,C 0.0631,E1 0.628,E2 462.252} C_DIS
LIN {X 134.6136,Y -36.1831,Z 192,A -7.2259,B 0.4692,C 0.0595,E1 0.629,E2 460.8206} C_DIS
LIN {X 135.5807,Y -32.3716,Z 192,A -5.8428,B 0.4697,C 0.0561,E1 0.6299,E2 459.4691} C_DIS
LIN {X 136.4371,Y -28.5567,Z 192,A -4.8899,B 0.4699,C 0.0545,E1 0.6304,E2 458.6062} C_DIS
LIN {X 137.3359,Y -23.8607,Z 192,A -3.2127,B 0.4703,C 0.0503,E1 0.6312,E2 456.9675} C_DIS
LIN {X 138.0134,Y -19.5534,Z 192,A -1.9435,B 0.4706,C 0.0475,E1 0.6317,E2 455.7689} C_DIS
LIN {X 138.4308,Y -16.3389,Z 192,A -0.8806,B 0.4709,C 0.045,E1 0.6321,E2 454.7418} C_DIS
LIN {X 138.8778,Y -11.9596,Z 192,A 0.5088,B 0.4712,C 0.0417,E1 0.6324,E2 453.4083} C_DIS
LIN {X 139.141,Y -8.3588,Z 192,A 1.655,B 0.4714,C 0.039,E1 0.6326,E2 452.3067} C_DIS
LIN {X 139.3276,Y -4.2436,Z 192,A 3.006,B 0.4716,C 0.0358,E1 0.6328,E2 451.0006} C_DIS
LIN {X 139.3947,Y -0.1243,Z 192,A 4.4075,B 0.4719,C 0.0323,E1 0.6328,E2 449.6371} C_DIS
LIN {X 139.3394,Y 3.8203,Z 192,A 5.5738,B 0.4721,C 0.0297,E1 0.6328,E2 448.53} C_DIS
LIN {X 139.1528,Y 8.1669,Z 192,A 7.0007,B 0.4723,C 0.0262,E1 0.6325,E2 447.1496} C_DIS
LIN {X 138.8567,Y 12.2098,Z 192,A 8.1984,B 0.4724,C 0.0236,E1 0.6323,E2 446.0122} C_DIS
LIN {X 138.5248,Y 15.533,Z 192,A 9.2595,B 0.4725,C 0.021,E1 0.632,E2 444.9908} C_DIS
LIN {X 138.1379,Y 18.6612,Z 192,A 10.3814,B 0.4726,C 0.0182,E1 0.6316,E2 443.8907} C_DIS
LIN {X 136.9262,Y 26.0997,Z 192,A 12.4898,B 0.4728,C 0.0137,E1 0.6307,E2 441.907} C_DIS
LIN {X 136.2976,Y 29.206,Z 192,A 13.7567,B 0.4728,C 0.0102,E1 0.63,E2 440.644} C_DIS
LIN {X 135.4313,Y 32.9914,Z 192,A 14.9795,B 0.4729,C 0.0074,E1 0.6292,E2 439.4675} C_DIS
LIN {X 134.1535,Y 37.8534,Z 192,A 16.5766,B 0.4729,C 0.0036,E1 0.6281,E2 437.9281} C_DIS
LIN {X 133.2162,Y 41.0297,Z 192,A 17.6079,B 0.4729,C 0.0013,E1 0.6273,E2 436.937} C_DIS
LIN {X 132.1757,Y 44.2671,Z 192,A 18.7183,B 0.4729,C -0.0014,E1 0.6263,E2 435.8615} C_DIS
LIN {X 130.9939,Y 47.6515,Z 192,A 19.8955,B 0.4729,C -0.0042,E1 0.6253,E2 434.7199} C_DIS
LIN {X 129.7206,Y 51.0174,Z 192,A 21.0148,B 0.4729,C -0.0067,E1 0.6242,E2 433.6439} C_DIS
LIN {X 128.4502,Y 54.1356,Z 192,A 22.0812,B 0.4729,C -0.0092,E1 0.6231,E2 432.6152} C_DIS
LIN {X 126.3456,Y 58.8801,Z 192,A 23.7028,B 0.4729,C -0.0128,E1 0.6213,E2 431.054} C_DIS
LIN {X 124.6065,Y 62.4807,Z 192,A 25.0421,B 0.4727,C -0.016,E1 0.6197,E2 429.7504} C_DIS
LIN {X 123.3792,Y 64.865,Z 192,A 25.8712,B 0.4727,C -0.0178,E1 0.6186,E2 428.9529} C_DIS
LIN {X 121.3906,Y 68.5189,Z 192,A 27.2894,B 0.4725,C -0.0212,E1 0.6167,E2 427.5685} C_DIS
LIN {X 119.1608,Y 72.3272,Z 192,A 28.747,B 0.4724,C -0.0245,E1 0.6147,E2 426.1518} C_DIS
LIN {X 116.7074,Y 76.2233,Z 192,A 30.22,B 0.4722,C -0.0278,E1 0.6125,E2 424.7267} C_DIS
LIN {X 114.189,Y 79.9469,Z 192,A 31.6878,B 0.472,C -0.031,E1 0.6102,E2 423.3018} C_DIS
LIN {X 111.5491,Y 83.5908,Z 192,A 33.1554,B 0.4718,C -0.0342,E1 0.6078,E2 421.8769} C_DIS
LIN {X 106.2142,Y 90.2718,Z 192,A 35.77,B 0.4713,C -0.0396,E1 0.6034,E2 419.3619} C_DIS
LIN {X 103.8016,Y 93.036,Z 192,A 37.1247,B 0.4711,C -0.0427,E1 0.6009,E2 418.0239} C_DIS
LIN {X 100.8057,Y 96.2739,Z 192,A 38.5942,B 0.4708,C -0.0458,E1 0.5981,E2 416.5917} C_DIS
LIN {X 97.4969,Y 99.6235,Z 192,A 40.879,B 0.4702,C -0.0515,E1 0.5933,E2 414.2688} C_DIS
LIN {X 92.0941,Y 104.6385,Z 192,A 42.5812,B 0.4699,C -0.0539,E1 0.59,E2 412.7094} C_DIS
LIN {X 88.4825,Y 107.7099,Z 192,A 44.1709,B 0.4695,C -0.0571,E1 0.5866,E2 411.1575} C_DIS
LIN {X 84.9257,Y 110.5358,Z 192,A 45.6273,B 0.4692,C -0.0598,E1 0.5834,E2 409.7439} C_DIS
LIN {X 81.4228,Y 113.1413,Z 192,A 47.1327,B 0.4688,C -0.0627,E1 0.58,E2 408.2684} C_DIS
LIN {X 77.6359,Y 115.7722,Z 192,A 48.6673,B 0.4684,C -0.0656,E1 0.5765,E2 406.7708} C_DIS
LIN {X 73.9057,Y 118.1884,Z 192,A 50.1473,B 0.4681,C -0.0682,E1 0.573,E2 405.3261} C_DIS
LIN {X 70.1493,Y 120.4561,Z 192,A 51.6538,B 0.4676,C -0.0709,E1 0.5693,E2 403.8495} C_DIS
LIN {X 66.2279,Y 122.6557,Z 192,A 53.1326,B 0.4673,C -0.0734,E1 0.5657,E2 402.4076} C_DIS
LIN {X 63.2269,Y 124.2266,Z 192,A 54.5666,B 0.4668,C -0.0762,E1 0.562,E2 400.9695} C_DIS
LIN {X 59.6253,Y 125.996,Z 192,A 55.3015,B 0.4668,C -0.0766,E1 0.5603,E2 400.3243} C_DIS
LIN {X 56.7138,Y 127.3322,Z 192,A 56.7047,B 0.4663,C -0.0793,E1 0.5566,E2 398.913} C_DIS
LIN {X 53.4714,Y 128.7276,Z 192,A 57.9109,B 0.466,C -0.0812,E1 0.5534,E2 397.7305} C_DIS
LIN {X 50.4214,Y 129.9523,Z 192,A 59.1029,B 0.4656,C -0.0831,E1 0.5502,E2 396.5541} C_DIS
LIN {X 46.0995,Y 131.5484,Z 192,A 60.7168,B 0.4652,C -0.0855,E1 0.5459,E2 394.9671} C_DIS
LIN {X 42.5746,Y 132.7304,Z 192,A 61.9407,B 0.4649,C -0.0872,E1 0.5426,E2 393.7722} C_DIS
LIN {X 36.9926,Y 134.3943,Z 192,A 63.9757,B 0.4643,C -0.09,E1 0.537,E2 391.7713} C_DIS
LIN {X 33.2993,Y 135.3571,Z 192,A 65.4211,B 0.464,C -0.0921,E1 0.533,E2 390.3377} C_DIS
LIN {X 26.5335,Y 136.8433,Z 192,A 67.64,B 0.4634,C -0.0946,E1 0.5268,E2 388.177} C_DIS
LIN {X 22.0285,Y 137.6417,Z 192,A 69.3897,B 0.463,C -0.0968,E1 0.5218,E2 386.4398} C_DIS
LIN {X 19.4541,Y 138.0276,Z 192,A 70.3788,B 0.4627,C -0.098,E1 0.5189,E2 385.4582} C_DIS
LIN {X 15.2916,Y 138.5508,Z 192,A 71.9344,B 0.4624,C -0.0997,E1 0.5144,E2 383.9183} C_DIS
LIN {X 11.6141,Y 138.907,Z 192,A 73.2631,B 0.4621,C -0.101,E1 0.5106,E2 382.6069} C_DIS
LIN {X 7.9984,Y 139.1632,Z 192,A 74.5422,B 0.4618,C -0.1022,E1 0.5069,E2 381.3471} C_DIS
LIN {X 4.356,Y 139.3245,Z 192,A 75.9841,B 0.4615,C -0.1037,E1 0.5027,E2 379.9107} C_DIS
LIN {X 0.1943,Y 139.3928,Z 192,A 77.4224,B 0.4612,C -0.1048,E1 0.4985,E2 378.4968} C_DIS
LIN {X -3.2616,Y 139.3549,Z 192,A 78.8778,B 0.4609,C -0.1061,E1 0.4942,E2 377.0389} C_DIS
LIN {X -7.2181,Y 139.2049,Z 192,A 80.2469,B 0.4607,C -0.107,E1 0.4902,E2 375.6928} C_DIS
LIN {X -11.2598,Y 138.9369,Z 192,A 81.8572,B 0.4605,C -0.1081,E1 0.4855,E2 374.0878} C_DIS
LIN {X -18.0822,Y 138.2138,Z 192,A 84.4669,B 0.4601,C -0.1096,E1 0.4779,E2 371.4974} C_DIS
LIN {X -26.4375,Y 136.8617,Z 192,A 88.2365,B 0.4596,C -0.1116,E1 0.4668,E2 367.7043} C_DIS
LIN {X -30.9741,Y 135.9065,Z 192,A 89.2498,B 0.4597,C -0.1114,E1 0.4641,E2 366.7678} C_DIS
LIN {X -30.9741,Y 135.9065,Z 192,A 89.2489,B 0.4597,C -0.1114,E1 0.4641,E2 366.7688} C_DIS
LIN {X -34.5652,Y 135.0381,Z 192,A 90.9466,B 0.4595,C -0.112,E1 0.4592,E2 365.0567} C_DIS
LIN {X -37.7202,Y 134.1908,Z 192,A 92.3328,B 0.4595,C -0.1123,E1 0.4552,E2 363.6675} C_DIS
LIN {X -41.031,Y 133.2158,Z 192,A 93.6999,B 0.4595,C -0.1125,E1 0.4513,E2 362.3053} C_DIS
LIN {X -44.4967,Y 132.0992,Z 192,A 95.2051,B 0.4594,C -0.1126,E1 0.4471,E2 360.8001} C_DIS
LIN {X -47.6758,Y 130.9852,Z 192,A 96.5481,B 0.4594,C -0.1126,E1 0.4434,E2 359.4611} C_DIS
LIN {X -50.4971,Y 129.9229,Z 192,A 97.8626,B 0.4594,C -0.1126,E1 0.4397,E2 358.1409} C_DIS
LIN {X -56.3622,Y 127.4895,Z 192,A 100.3909,B 0.4595,C -0.1121,E1 0.4328,E2 355.6207} C_DIS
LIN {X -59.0492,Y 126.2674,Z 192,A 101.9048,B 0.4595,C -0.1119,E1 0.4287,E2 354.0819} C_DIS
LIN {X -62.3429,Y 124.6749,Z 192,A 103.2992,B 0.4597,C -0.1114,E1 0.425,E2 352.6976} C_DIS
LIN {X -65.5693,Y 123.0094,Z 192,A 105.0107,B 0.4598,C -0.1108,E1 0.4204,E2 350.9682} C_DIS
LIN {X -70.7316,Y 120.1146,Z 192,A 108.4111,B 0.4601,C -0.1096,E1 0.4115,E2 347.4849} C_DIS
LIN {X -76.1706,Y 116.7416,Z 192,A 110.319,B 0.4605,C -0.1078,E1 0.4069,E2 345.6413} C_DIS
LIN {X -82.2843,Y 112.5159,Z 192,A 113.4759,B 0.4611,C -0.1054,E1 0.3993,E2 342.4773} C_DIS
LIN {X -84.6675,Y 110.7334,Z 192,A 115.1249,B 0.4614,C -0.1042,E1 0.3953,E2 340.7918} C_DIS
LIN {X -88.2213,Y 107.9234,Z 192,A 117.2528,B 0.4618,C -0.1022,E1 0.3904,E2 338.6414} C_DIS
LIN {X -91.8496,Y 104.8532,Z 192,A 119.4841,B 0.4623,C -0.0999,E1 0.3854,E2 336.3865} C_DIS
LIN {X -94.988,Y 102.0183,Z 192,A 121.4874,B 0.4628,C -0.0977,E1 0.381,E2 334.3604} C_DIS
LIN {X -98.122,Y 99.0079,Z 192,A 123.619,B 0.4633,C -0.0951,E1 0.3765,E2 332.1984} C_DIS
LIN {X -101.3419,Y 95.7094,Z 192,A 125.8256,B 0.4639,C -0.0923,E1 0.3719,E2 329.9643} C_DIS
LIN {X -104.2757,Y 92.5046,Z 192,A 128.0338,B 0.4645,C -0.0892,E1 0.3675,E2 327.718} C_DIS
LIN {X -107.2734,Y 89.0106,Z 192,A 130.2982,B 0.4651,C -0.0859,E1 0.3632,E2 325.4198} C_DIS
LIN {X -110.0542,Y 85.5487,Z 192,A 133.6264,B 0.466,C -0.0811,E1 0.3571,E2 321.948} C_DIS
LIN {X -113.9955,Y 80.2216,Z 192,A 136.0036,B 0.4667,C -0.0767,E1 0.3531,E2 319.6062} C_DIS
LIN {X -116.6006,Y 76.3862,Z 192,A 138.4186,B 0.4674,C -0.0724,E1 0.3492,E2 317.1424} C_DIS
LIN {X -119.0295,Y 72.5438,Z 192,A 141.1268,B 0.4682,C -0.0675,E1 0.3449,E2 314.3513} C_DIS
LIN {X -120.7344,Y 69.6686,Z 192,A 142.4679,B 0.4685,C -0.0647,E1 0.343,E2 313.0143} C_DIS
LIN {X -122.593,Y 66.3446,Z 192,A 144.7583,B 0.4691,C -0.0603,E1 0.3398,E2 310.6509} C_DIS
LIN {X -124.5073,Y 62.6755,Z 192,A 146.8254,B 0.4697,C -0.056,E1 0.337,E2 308.5467} C_DIS
LIN {X -126.2293,Y 59.1316,Z 192,A 149.1248,B 0.4702,C -0.0513,E1 0.3341,E2 306.1769} C_DIS
LIN {X -130.1659,Y 49.8721,Z 192,A 154.5125,B 0.4714,C -0.0393,E1 0.3281,E2 300.6572} C_DIS
LIN {X -130.1659,Y 49.8721,Z 192,A 154.511,B 0.4714,C -0.0393,E1 0.3281,E2 300.6589} C_DIS
LIN {X -131.692,Y 45.6852,Z 192,A 157.2767,B 0.4718,C -0.0331,E1 0.3253,E2 297.7911} C_DIS
LIN {X -132.857,Y 42.1783,Z 192,A 159.3272,B 0.4722,C -0.0283,E1 0.3235,E2 295.6817} C_DIS
LIN {X -133.8691,Y 38.8473,Z 192,A 161.3386,B 0.4724,C -0.0235,E1 0.3218,E2 293.6051} C_DIS
LIN {X -135.3665,Y 33.2601,Z 192,A 164.5511,B 0.4727,C -0.0157,E1 0.3195,E2 290.2975} C_DIS
LIN {X -135.3665,Y 33.2601,Z 192,A 164.5502,B 0.4727,C -0.0157,E1 0.3195,E2 290.2985} C_DIS
LIN {X -136.3882,Y 28.7861,Z 192,A 167.3177,B 0.4729,C -0.0089,E1 0.3177,E2 287.4284} C_DIS
LIN {X -136.9866,Y 25.7837,Z 192,A 169.3306,B 0.4729,C -0.004,E1 0.3166,E2 285.3257} C_DIS
LIN {X -137.8909,Y 20.4106,Z 192,A 173.7598,B 0.4729,C 0.0067,E1 0.3147,E2 280.6276} C_DIS
LIN {X -138.706,Y 13.8168,Z 192,A 176.1475,B 0.4729,C 0.0135,E1 0.3139,E2 278.2845} C_DIS
LIN {X -138.982,Y 10.6921,Z 192,A 179.4193,B 0.4725,C 0.0212,E1 0.3132,E2 274.7605} C_DIS
LIN {X -139.3183,Y 4.5792,Z 192,A -178.2149,B 0.4722,C 0.0279,E1 0.3129,E2 272.4158} C_DIS
LIN {X -139.3799,Y -1.8693,Z 192,A -174.504,B 0.4715,C 0.0375,E1 0.3129,E2 268.5676} C_DIS
LIN {X -139.3799,Y -1.8693,Z 192,A -174.5051,B 0.4715,C 0.0375,E1 0.3129,E2 268.5689} C_DIS
LIN {X -139.0966,Y -9.0785,Z 192,A -169.6734,B 0.4704,C 0.0495,E1 0.3135,E2 263.4887} C_DIS
LIN {X -139.0966,Y -9.0785,Z 192,A -169.6748,B 0.4704,C 0.0495,E1 0.3135,E2 263.4902} C_DIS
LIN {X -138.7597,Y -13.2583,Z 192,A -167.4988,B 0.4698,C 0.0552,E1 0.3141,E2 261.2533} C_DIS
LIN {X -138.3807,Y -16.7588,Z 192,A -165.4571,B 0.4691,C 0.0603,E1 0.3147,E2 259.1305} C_DIS
LIN {X -137.9556,Y -19.9579,Z 192,A -162.9682,B 0.4683,C 0.0662,E1 0.3158,E2 256.48} C_DIS
LIN {X -137.357,Y -23.7421,Z 192,A -161.1887,B 0.4677,C 0.0708,E1 0.3166,E2 254.6724} C_DIS
LIN {X -136.6317,Y -27.6005,Z 192,A -158.8601,B 0.4668,C 0.0764,E1 0.3179,E2 252.2431} C_DIS
LIN {X -135.8806,Y -31.0873,Z 192,A -156.8859,B 0.466,C 0.0812,E1 0.3192,E2 250.1969} C_DIS
LIN {X -135.027,Y -34.6088,Z 192,A -154.8401,B 0.4651,C 0.086,E1 0.3206,E2 248.0715} C_DIS
LIN {X -134.1396,Y -37.9034,Z 192,A -152.8059,B 0.4642,C 0.0907,E1 0.3222,E2 245.9461} C_DIS
LIN {X -133.1269,Y -41.3215,Z 192,A -150.7604,B 0.4633,C 0.0954,E1 0.324,E2 243.8163} C_DIS
LIN {X -130.4198,Y -49.2008,Z 192,A -146.0586,B 0.461,C 0.1057,E1 0.3286,E2 238.9268} C_DIS
LIN {X -130.4198,Y -49.2008,Z 192,A -146.0596,B 0.461,C 0.1057,E1 0.3286,E2 238.928} C_DIS
LIN {X -129.2257,Y -52.2555,Z 192,A -144.1418,B 0.4601,C 0.1097,E1 0.3306,E2 236.9254} C_DIS
LIN {X -127.5411,Y -56.2468,Z 192,A -141.8973,B 0.4589,C 0.1145,E1 0.3332,E2 234.6117} C_DIS
LIN {X -126.4709,Y -58.6091,Z 192,A -140.3443,B 0.4582,C 0.1175,E1 0.3352,E2 232.9852} C_DIS
LIN {X -124.8113,Y -62.0663,Z 192,A -138.2729,B 0.4571,C 0.1216,E1 0.3379,E2 230.839} C_DIS
LIN {X -122.6648,Y -66.2109,Z 192,A -135.6837,B 0.4558,C 0.1264,E1 0.3415,E2 228.1476} C_DIS
LIN {X -120.4223,Y -70.2077,Z 192,A -133.1946,B 0.4545,C 0.1309,E1 0.3452,E2 225.5656} C_DIS
LIN {X -118.0341,Y -74.1518,Z 192,A -130.7892,B 0.4533,C 0.135,E1 0.3489,E2 223.0815} C_DIS
LIN {X -115.5963,Y -77.8976,Z 192,A -128.5503,B 0.4522,C 0.1388,E1 0.3526,E2 220.7803} C_DIS
LIN {X -113.1341,Y -81.433,Z 192,A -126.2485,B 0.4511,C 0.1423,E1 0.3566,E2 218.3957} C_DIS
LIN {X -109.6389,Y -86.08,Z 192,A -123.4657,B 0.4497,C 0.1466,E1 0.3616,E2 215.5516} C_DIS
LIN {X -107.1307,Y -89.183,Z 192,A -121.3285,B 0.4488,C 0.1494,E1 0.3657,E2 213.3361} C_DIS
LIN {X -104.6123,Y -92.1238,Z 192,A -119.4155,B 0.4479,C 0.1519,E1 0.3694,E2 211.3723} C_DIS
LIN {X -101.5501,Y -95.4887,Z 192,A -117.2088,B 0.447,C 0.1547,E1 0.3739,E2 209.1122} C_DIS
LIN {X -96.0379,Y -101.0313,Z 192,A -113.765,B 0.4455,C 0.1588,E1 0.3811,E2 205.6319} C_DIS
LIN {X -92.4465,Y -104.327,Z 192,A -111.085,B 0.4447,C 0.1611,E1 0.3872,E2 202.8437} C_DIS
LIN {X -89.4455,Y -106.9112,Z 192,A -109.3548,B 0.4441,C 0.1628,E1 0.3911,E2 201.097} C_DIS
LIN {X -85.9696,Y -109.7256,Z 192,A -107.2803,B 0.4435,C 0.1645,E1 0.396,E2 198.9844} C_DIS
LIN {X -82.3181,Y -112.4911,Z 192,A -105.1799,B 0.4429,C 0.166,E1 0.401,E2 196.8487} C_DIS
LIN {X -78.7086,Y -115.0454,Z 192,A -103.1889,B 0.4424,C 0.1673,E1 0.4059,E2 194.8293} C_DIS
LIN {X -74.8072,Y -117.6202,Z 192,A -101.1364,B 0.442,C 0.1685,E1 0.4111,E2 192.7553} C_DIS
LIN {X -70.9697,Y -119.9747,Z 192,A -99.1216,B 0.4416,C 0.1695,E1 0.4162,E2 190.7135} C_DIS
LIN {X -67.0992,Y -122.1815,Z 192,A -97.2146,B 0.4413,C 0.1703,E1 0.4212,E2 188.7938} C_DIS
LIN {X -62.9674,Y -124.3587,Z 192,A -95.2944,B 0.441,C 0.171,E1 0.4263,E2 186.8729} C_DIS
LIN {X -59.6756,Y -125.9719,Z 192,A -93.7259,B 0.4409,C 0.1714,E1 0.4305,E2 185.2939} C_DIS
LIN {X -55.7287,Y -127.767,Z 192,A -91.8686,B 0.4407,C 0.1717,E1 0.4355,E2 183.4238} C_DIS
LIN {X -52.1105,Y -129.2842,Z 192,A -90.2484,B 0.4407,C 0.1719,E1 0.44,E2 181.8018} C_DIS
LIN {X -48.6535,Y -130.6247,Z 192,A -88.7382,B 0.4407,C 0.1719,E1 0.4442,E2 180.2932} C_DIS
LIN {X -44.7528,Y -132.0139,Z 192,A -86.5008,B 0.4409,C 0.1712,E1 0.4507,E2 177.9681} C_DIS
LIN {X -40.084,Y -133.5057,Z 192,A -85.0909,B 0.4407,C 0.1718,E1 0.4544,E2 176.6555} C_DIS
LIN {X -37.1697,Y -134.3447,Z 192,A -83.7471,B 0.4409,C 0.1714,E1 0.4583,E2 175.2953} C_DIS
LIN {X -31.1066,Y -135.8762,Z 192,A -81.3025,B 0.4411,C 0.1708,E1 0.4653,E2 172.8698} C_DIS
LIN {X -26.6737,Y -136.8165,Z 192,A -79.4827,B 0.4413,C 0.1702,E1 0.4706,E2 171.056} C_DIS
LIN {X -22.7785,Y -137.5179,Z 192,A -78.0172,B 0.4415,C 0.1697,E1 0.4748,E2 169.6156} C_DIS
LIN {X -19.1285,Y -138.0741,Z 192,A -76.494,B 0.4418,C 0.1689,E1 0.4792,E2 168.0906} C_DIS
LIN {X -14.7224,Y -138.6121,Z 192,A -74.8761,B 0.4421,C 0.1682,E1 0.4839,E2 166.505} C_DIS
LIN {X -10.8632,Y -138.9695,Z 192,A -73.3006,B 0.4425,C 0.1671,E1 0.4885,E2 164.9314} C_DIS
LIN {X -7.0525,Y -139.2132,Z 192,A -71.9335,B 0.4428,C 0.1663,E1 0.4925,E2 163.5961} C_DIS
LIN {X -3.4536,Y -139.3496,Z 192,A -70.6117,B 0.4431,C 0.1655,E1 0.4963,E2 162.2988} C_DIS
LIN {X 0.0758,Y -139.3935,Z 192,A -69.1485,B 0.4436,C 0.1642,E1 0.5006,E2 160.8327} C_DIS
LIN {X 0.0758,Y -139.3935,Z 192,A -69.1485,B 0.4436,C 0.1642,E1 0.5006,E2 160.8327} C_DIS
Enddeposition()
LIN {X 1.0037,Y -140.2868,Z 192,A -70.0449,B 0.4632,C 0.1675,E1 0.518,E2 161.9438} C_DIS
Startdeposition()
$VEL.CP = VEL_PRINT
LIN {X -2.5481,Y -140.2677,Z 192,A -71.4398,B 0.4628,C 0.1686,E1 0.5139,E2 163.3307} C_DIS
LIN {X -7.0436,Y -140.1137,Z 192,A -73.1023,B 0.4625,C 0.1696,E1 0.5091,E2 164.9662} C_DIS
LIN {X -11.1985,Y -139.8442,Z 192,A -74.8089,B 0.462,C 0.1708,E1 0.5041,E2 166.6749} C_DIS
LIN {X -15.7672,Y -139.4037,Z 192,A -76.5519,B 0.4617,C 0.1716,E1 0.499,E2 168.3979} C_DIS
LIN {X -19.5206,Y -138.9261,Z 192,A -77.8464,B 0.4616,C 0.172,E1 0.4954,E2 169.6527} C_DIS
LIN {X -22.8802,Y -138.4122,Z 192,A -79.254,B 0.4613,C 0.1727,E1 0.4913,E2 171.0642} C_DIS
LIN {X -26.2781,Y -137.8073,Z 192,A -80.4872,B 0.4613,C 0.1729,E1 0.4878,E2 172.2697} C_DIS
LIN {X -30.0469,Y -137.0357,Z 192,A -82.6078,B 0.4607,C 0.1743,E1 0.4814,E2 174.4799} C_DIS
LIN {X -34.6267,Y -135.9499,Z 192,A -83.9898,B 0.4608,C 0.174,E1 0.4777,E2 175.7756} C_DIS
LIN {X -45.3998,Y -132.7424,Z 192,A -88.5759,B 0.4607,C 0.1744,E1 0.4647,E2 180.3632} C_DIS
LIN {X -45.3998,Y -132.7424,Z 192,A -88.5769,B 0.4607,C 0.1744,E1 0.4647,E2 180.3643} C_DIS
LIN {X -48.9451,Y -131.4754,Z 192,A -90.0435,B 0.4607,C 0.1742,E1 0.4607,E2 181.82} C_DIS
LIN {X -52.0278,Y -130.2867,Z 192,A -91.4522,B 0.4607,C 0.1742,E1 0.4568,E2 183.2389} C_DIS
LIN {X -54.9483,Y -129.0838,Z 192,A -92.8615,B 0.4608,C 0.174,E1 0.4529,E2 184.668} C_DIS
LIN {X -58.514,Y -127.5052,Z 192,A -94.4369,B 0.461,C 0.1736,E1 0.4487,E2 186.2412} C_DIS
LIN {X -62.3812,Y -125.6583,Z 192,A -96.2282,B 0.4612,C 0.173,E1 0.4439,E2 188.0396} C_DIS
LIN {X -66.6285,Y -123.4609,Z 192,A -98.3327,B 0.4614,C 0.1723,E1 0.4383,E2 190.1692} C_DIS
LIN {X -70.6546,Y -121.2022,Z 192,A -100.3222,B 0.4618,C 0.1714,E1 0.4332,E2 192.1759} C_DIS
LIN {X -74.2441,Y -119.0366,Z 192,A -102.1149,B 0.4622,C 0.1703,E1 0.4287,E2 193.982} C_DIS
LIN {X -77.542,Y -116.9157,Z 192,A -103.904,B 0.4626,C 0.1693,E1 0.4242,E2 195.8016} C_DIS
LIN {X -81.2132,Y -114.3961,Z 192,A -105.9212,B 0.4631,C 0.1679,E1 0.4193,E2 197.8511} C_DIS
LIN {X -84.9118,Y -111.6781,Z 192,A -107.9941,B 0.4636,C 0.1663,E1 0.4143,E2 199.956} C_DIS
LIN {X -88.4817,Y -108.8715,Z 192,A -110.0511,B 0.4643,C 0.1645,E1 0.4095,E2 202.0455} C_DIS
LIN {X -93.4229,Y -104.6618,Z 192,A -114.6301,B 0.4654,C 0.1614,E1 0.3989,E2 206.9302} C_DIS
LIN {X -100.5275,Y -97.8582,Z 192,A -117.7647,B 0.4671,C 0.1563,E1 0.3927,E2 209.9257} C_DIS
LIN {X -103.72,Y -94.4675,Z 192,A -119.9986,B 0.468,C 0.1535,E1 0.3882,E2 212.2119} C_DIS
LIN {X -107.2795,Y -90.4051,Z 192,A -122.6215,B 0.4692,C 0.1499,E1 0.3831,E2 214.9002} C_DIS
LIN {X -112.6479,Y -83.6204,Z 192,A -126.8927,B 0.4712,C 0.1436,E1 0.3753,E2 219.2866} C_DIS
LIN {X -115.2545,Y -79.9894,Z 192,A -129.134,B 0.4723,C 0.14,E1 0.3715,E2 221.5923} C_DIS
LIN {X -117.6824,Y -76.3723,Z 192,A -131.4121,B 0.4734,C 0.1362,E1 0.3677,E2 223.9473} C_DIS
LIN {X -120.1702,Y -72.3951,Z 192,A -133.7806,B 0.4745,C 0.132,E1 0.3641,E2 226.3851} C_DIS
LIN {X -122.215,Y -68.8869,Z 192,A -135.9951,B 0.4756,C 0.128,E1 0.3608,E2 228.6845} C_DIS
LIN {X -124.2998,Y -65.0452,Z 192,A -138.1475,B 0.4767,C 0.1238,E1 0.3578,E2 230.8924} C_DIS
LIN {X -125.6994,Y -62.2979,Z 192,A -139.8218,B 0.4776,C 0.1206,E1 0.3556,E2 232.6293} C_DIS
LIN {X -127.5672,Y -58.38,Z 192,A -142.1777,B 0.4787,C 0.1159,E1 0.3526,E2 235.0727} C_DIS
LIN {X -128.9139,Y -55.3412,Z 192,A -144.1537,B 0.4797,C 0.1119,E1 0.3503,E2 237.1409} C_DIS
LIN {X -130.6484,Y -51.1119,Z 192,A -146.5275,B 0.4809,C 0.1068,E1 0.3477,E2 239.5895} C_DIS
LIN {X -132.6831,Y -45.5708,Z 192,A -149.8544,B 0.4824,C 0.0995,E1 0.3444,E2 243.0507} C_DIS
LIN {X -134.0445,Y -41.3951,Z 192,A -152.0099,B 0.4834,C 0.0945,E1 0.3425,E2 245.2584} C_DIS
LIN {X -135.0567,Y -37.9617,Z 192,A -154.1151,B 0.4843,C 0.0897,E1 0.3408,E2 247.4565} C_DIS
LIN {X -135.9224,Y -34.7349,Z 192,A -156.0578,B 0.4852,C 0.0852,E1 0.3394,E2 249.482} C_DIS
LIN {X -136.7371,Y -31.3747,Z 192,A -157.851,B 0.4859,C 0.0808,E1 0.3382,E2 251.3291} C_DIS
LIN {X -137.4112,Y -28.2781,Z 192,A -159.7737,B 0.4866,C 0.0762,E1 0.337,E2 253.3405} C_DIS
LIN {X -137.992,Y -25.2973,Z 192,A -162.8366,B 0.4876,C 0.0696,E1 0.3354,E2 256.6575} C_DIS
LIN {X -139.0279,Y -18.7881,Z 192,A -165.4668,B 0.4886,C 0.0623,E1 0.3343,E2 259.2779} C_DIS
LIN {X -139.6049,Y -13.86,Z 192,A -168.4784,B 0.4895,C 0.0549,E1 0.3333,E2 262.4232} C_DIS
LIN {X -140.212,Y -4.7507,Z 192,A -173.4884,B 0.4908,C 0.042,E1 0.3325,E2 267.6033} C_DIS
LIN {X -140.212,Y -4.7507,Z 192,A -173.4893,B 0.4908,C 0.042,E1 0.3325,E2 267.6044} C_DIS
LIN {X -140.2543,Y 3.2557,Z 192,A -178.0765,B 0.4916,C 0.0302,E1 0.3325,E2 272.3629} C_DIS
LIN {X -140.2543,Y 3.2557,Z 192,A -178.078,B 0.4916,C 0.0302,E1 0.3325,E2 272.3646} C_DIS
LIN {X -139.9,Y 10.464,Z 192,A 177.5644,B 0.4922,C 0.0191,E1 0.3332,E2 276.9011} C_DIS
LIN {X -139.9,Y 10.464,Z 192,A 177.5629,B 0.4922,C 0.0191,E1 0.3332,E2 276.9028} C_DIS
LIN {X -139.4851,Y 15.0116,Z 192,A 174.403,B 0.4924,C 0.0113,E1 0.3341,E2 280.2232} C_DIS
LIN {X -139.0176,Y 18.8663,Z 192,A 171.7879,B 0.4925,C 0.0049,E1 0.3351,E2 282.963} C_DIS
LIN {X -138.2282,Y 23.9776,Z 192,A 169.5585,B 0.4925,C -0.0011,E1 0.3362,E2 285.2053} C_DIS
LIN {X -137.5573,Y 27.5598,Z 192,A 167.6075,B 0.4925,C -0.006,E1 0.3373,E2 287.2107} C_DIS
LIN {X -136.8319,Y 30.9597,Z 192,A 165.505,B 0.4925,C -0.0112,E1 0.3386,E2 289.393} C_DIS
LIN {X -135.2259,Y 37.3565,Z 192,A 161.9745,B 0.4922,C -0.0198,E1 0.3411,E2 293.0194} C_DIS
LIN {X -135.2259,Y 37.3565,Z 192,A 161.9734,B 0.4922,C -0.0198,E1 0.3411,E2 293.0206} C_DIS
LIN {X -134.2198,Y 40.8222,Z 192,A 159.8462,B 0.4919,C -0.0249,E1 0.3429,E2 295.2216} C_DIS
LIN {X -133.2085,Y 44.0108,Z 192,A 158.1111,B 0.4917,C -0.029,E1 0.3444,E2 296.9976} C_DIS
LIN {X -131.9742,Y 47.583,Z 192,A 155.8891,B 0.4914,C -0.0341,E1 0.3466,E2 299.2944} C_DIS
LIN {X -130.9264,Y 50.3966,Z 192,A 154.3807,B 0.4911,C -0.0376,E1 0.3481,E2 300.8332} C_DIS
LIN {X -129.9813,Y 52.7856,Z 192,A 151.8899,B 0.4907,C -0.0426,E1 0.351,E2 303.479} C_DIS
LIN {X -127.9614,Y 57.5088,Z 192,A 150.0791,B 0.4903,C -0.047,E1 0.353,E2 305.2581} C_DIS
LIN {X -125.839,Y 62.0149,Z 192,A 147.2767,B 0.4897,C -0.0529,E1 0.3565,E2 308.1406} C_DIS
LIN {X -124.3604,Y 64.9299,Z 192,A 145.5287,B 0.4893,C -0.0565,E1 0.3588,E2 309.9308} C_DIS
LIN {X -122.4283,Y 68.5073,Z 192,A 143.5259,B 0.4888,C -0.0605,E1 0.3616,E2 311.9681} C_DIS
LIN {X -118.8035,Y 74.617,Z 192,A 139.482,B 0.4878,C -0.068,E1 0.3678,E2 316.1259} C_DIS
LIN {X -118.8035,Y 74.617,Z 192,A 139.4807,B 0.4878,C -0.068,E1 0.3678,E2 316.1273} C_DIS
LIN {X -114.9132,Y 80.48,Z 192,A 135.301,B 0.4868,C -0.0751,E1 0.3747,E2 320.4329} C_DIS
LIN {X -112.2789,Y 84.1157,Z 192,A 133.442,B 0.4863,C -0.0784,E1 0.3779,E2 322.2933} C_DIS
LIN {X -109.1006,Y 88.1984,Z 192,A 131.0184,B 0.4856,C -0.0824,E1 0.3823,E2 324.7453} C_DIS
LIN {X -106.3015,Y 91.5525,Z 192,A 128.8049,B 0.4851,C -0.0856,E1 0.3866,E2 326.9983} C_DIS
LIN {X -103.2703,Y 94.9585,Z 192,A 126.5624,B 0.4845,C -0.0888,E1 0.391,E2 329.275} C_DIS
LIN {X -100.0575,Y 98.3381,Z 192,A 124.3566,B 0.484,C -0.0917,E1 0.3955,E2 331.5076} C_DIS
LIN {X -96.9107,Y 101.4405,Z 192,A 122.2304,B 0.4835,C -0.0943,E1 0.4,E2 333.6621} C_DIS
LIN {X -93.7891,Y 104.3338,Z 192,A 120.1612,B 0.483,C -0.0966,E1 0.4045,E2 335.7602} C_DIS
LIN {X -90.4894,Y 107.2088,Z 192,A 118.1336,B 0.4826,C -0.0988,E1 0.4091,E2 337.8084} C_DIS
LIN {X -87.0191,Y 110.0443,Z 192,A 116.0437,B 0.4821,C -0.1008,E1 0.4139,E2 339.9204} C_DIS
LIN {X -83.4884,Y 112.7461,Z 192,A 114.2357,B 0.4818,C -0.1025,E1 0.4181,E2 341.7268} C_DIS
LIN {X -80.6677,Y 114.7807,Z 192,A 112.3228,B 0.4815,C -0.1038,E1 0.4228,E2 343.682} C_DIS
LIN {X -76.2328,Y 117.773,Z 192,A 110.164,B 0.4811,C -0.1055,E1 0.4281,E2 345.8375} C_DIS
LIN {X -72.3042,Y 120.2252,Z 192,A 108.0276,B 0.4809,C -0.1067,E1 0.4335,E2 347.9942} C_DIS
LIN {X -67.3191,Y 123.0855,Z 192,A 105.5551,B 0.4806,C -0.108,E1 0.4399,E2 350.4763} C_DIS
LIN {X -63.9382,Y 124.8732,Z 192,A 104.1175,B 0.4804,C -0.1087,E1 0.4436,E2 351.9024} C_DIS
LIN {X -60.8553,Y 126.4045,Z 192,A 102.5359,B 0.4804,C -0.1091,E1 0.4478,E2 353.4985} C_DIS
LIN {X -58.4741,Y 127.5237,Z 192,A 101.3363,B 0.4803,C -0.1094,E1 0.4511,E2 354.7082} C_DIS
LIN {X -52.8571,Y 129.9525,Z 192,A 98.8599,B 0.4801,C -0.1099,E1 0.4578,E2 357.1816} C_DIS
LIN {X -49.5004,Y 131.2674,Z 192,A 97.5949,B 0.4801,C -0.1102,E1 0.4612,E2 358.4281} C_DIS
LIN {X -46.5253,Y 132.3522,Z 192,A 96.0463,B 0.4801,C -0.1102,E1 0.4656,E2 359.9981} C_DIS
LIN {X -43.2164,Y 133.4691,Z 192,A 94.5833,B 0.4801,C -0.11,E1 0.4697,E2 361.4636} C_DIS
LIN {X -39.8531,Y 134.5113,Z 192,A 93.2538,B 0.4801,C -0.11,E1 0.4734,E2 362.7832} C_DIS
LIN {X -36.2613,Y 135.523,Z 192,A 91.8572,B 0.4801,C -0.1098,E1 0.4774,E2 364.1681} C_DIS
LIN {X -33.426,Y 136.2512,Z 192,A 90.696,B 0.4802,C -0.1096,E1 0.4807,E2 365.326} C_DIS
LIN {X -30.2588,Y 136.9899,Z 192,A 89.2097,B 0.4804,C -0.109,E1 0.485,E2 366.8253} C_DIS
LIN {X -26.52,Y 137.7611,Z 192,A 87.9076,B 0.4804,C -0.1087,E1 0.4887,E2 368.1047} C_DIS
LIN {X -23.7078,Y 138.2741,Z 192,A 86.469,B 0.4806,C -0.1079,E1 0.493,E2 369.5661} C_DIS
LIN {X -17.5559,Y 139.1893,Z 192,A 84.231,B 0.4808,C -0.107,E1 0.4994,E2 371.7772} C_DIS
LIN {X -13.9049,Y 139.6006,Z 192,A 82.8173,B 0.481,C -0.1061,E1 0.5035,E2 373.1828} C_DIS
LIN {X -10.1998,Y 139.9193,Z 192,A 81.4398,B 0.4812,C -0.1053,E1 0.5075,E2 374.5473} C_DIS
LIN {X -5.8049,Y 140.1709,Z 192,A 79.7623,B 0.4814,C -0.1041,E1 0.5124,E2 376.2137} C_DIS
LIN {X -1.8416,Y 140.2794,Z 192,A 78.2274,B 0.4817,C -0.1029,E1 0.5169,E2 377.7407} C_DIS
LIN {X 2.319,Y 140.2715,Z 192,A 76.7316,B 0.4819,C -0.1017,E1 0.5212,E2 379.218} C_DIS
LIN {X 6.6413,Y 140.1339,Z 192,A 75.1751,B 0.4822,C -0.1004,E1 0.5257,E2 380.7553} C_DIS
LIN {X 10.1782,Y 139.9209,Z 192,A 73.869,B 0.4825,C -0.0991,E1 0.5295,E2 382.0484} C_DIS
LIN {X 14.2531,Y 139.5667,Z 192,A 72.3464,B 0.4828,C -0.0976,E1 0.5339,E2 383.5574} C_DIS
LIN {X 17.7551,Y 139.1632,Z 192,A 71.0014,B 0.4831,C -0.0961,E1 0.5378,E2 384.8934} C_DIS
LIN {X 22.1415,Y 138.5339,Z 192,A 69.47,B 0.4834,C -0.0944,E1 0.5421,E2 386.3991} C_DIS
LIN {X 26.0802,Y 137.8452,Z 192,A 68.2643,B 0.4837,C -0.0933,E1 0.5455,E2 387.5652} C_DIS
LIN {X 30.5397,Y 136.9271,Z 192,A 66.3429,B 0.4842,C -0.0906,E1 0.551,E2 389.4919} C_DIS
LIN {X 34.4488,Y 135.9951,Z 192,A 64.0998,B 0.4849,C -0.0867,E1 0.5575,E2 391.7893} C_DIS
LIN {X 41.7874,Y 133.9244,Z 192,A 62.229,B 0.4852,C -0.085,E1 0.5624,E2 393.5452} C_DIS
LIN {X 46.0051,Y 132.5325,Z 192,A 60.8529,B 0.4855,C -0.0832,E1 0.566,E2 394.8795} C_DIS
LIN {X 48.8966,Y 131.4936,Z 192,A 59.7247,B 0.4858,C -0.0815,E1 0.569,E2 395.9954} C_DIS
LIN {X 51.7812,Y 130.3862,Z 192,A 58.5574,B 0.4861,C -0.0796,E1 0.5722,E2 397.1535} C_DIS
LIN {X 55.4089,Y 128.8847,Z 192,A 57.3179,B 0.4864,C -0.0778,E1 0.5754,E2 398.3577} C_DIS
LIN {X 58.5602,Y 127.4839,Z 192,A 56.1076,B 0.4867,C -0.0758,E1 0.5785,E2 399.5485} C_DIS
LIN {X 62.5229,Y 125.5884,Z 192,A 54.496,B 0.4871,C -0.073,E1 0.5826,E2 401.1421} C_DIS
LIN {X 66.7943,Y 123.3718,Z 192,A 52.8739,B 0.4875,C -0.0703,E1 0.5867,E2 402.7302} C_DIS
LIN {X 70.6763,Y 121.1896,Z 192,A 51.4306,B 0.4879,C -0.0679,E1 0.5902,E2 404.136} C_DIS
LIN {X 74.3875,Y 118.9473,Z 192,A 49.9158,B 0.4882,C -0.0651,E1 0.5938,E2 405.6249} C_DIS
LIN {X 78.2751,Y 116.4263,Z 192,A 48.3402,B 0.4886,C -0.0622,E1 0.5975,E2 407.1684} C_DIS
LIN {X 82.0371,Y 113.8065,Z 192,A 46.8008,B 0.489,C -0.0593,E1 0.601,E2 408.6737} C_DIS
LIN {X 85.6105,Y 111.1436,Z 192,A 45.3094,B 0.4893,C -0.0565,E1 0.6043,E2 410.1312} C_DIS
LIN {X 89.3813,Y 108.1336,Z 192,A 43.7261,B 0.4897,C -0.0534,E1 0.6078,E2 411.6742} C_DIS
LIN {X 92.9685,Y 105.0654,Z 192,A 42.3622,B 0.4899,C -0.051,E1 0.6106,E2 412.9786} C_DIS
LIN {X 96.6105,Y 101.7268,Z 192,A 40.4504,B 0.4903,C -0.0468,E1 0.6145,E2 414.8792} C_DIS
LIN {X 100.3702,Y 98.0193,Z 192,A 38.7928,B 0.4906,C -0.0435,E1 0.6178,E2 416.4835} C_DIS
LIN {X 103.5507,Y 94.6534,Z 192,A 37.2634,B 0.4909,C -0.0403,E1 0.6206,E2 417.9738} C_DIS
LIN {X 106.4391,Y 91.3927,Z 192,A 35.8606,B 0.4912,C -0.0373,E1 0.6232,E2 419.3356} C_DIS
LIN {X 109.8642,Y 87.2447,Z 192,A 34.0511,B 0.4914,C -0.0334,E1 0.6263,E2 421.1026} C_DIS
LIN {X 112.8221,Y 83.3858,Z 192,A 32.4866,B 0.4917,C -0.03,E1 0.6289,E2 422.6203} C_DIS
LIN {X 115.4094,Y 79.7668,Z 192,A 31.0441,B 0.4918,C -0.0268,E1 0.6312,E2 424.021} C_DIS
LIN {X 117.8823,Y 76.0644,Z 192,A 29.6262,B 0.492,C -0.0237,E1 0.6333,E2 425.3937} C_DIS
LIN {X 120.2097,Y 72.3297,Z 192,A 28.1868,B 0.4921,C -0.0205,E1 0.6354,E2 426.7924} C_DIS
LIN {X 122.4285,Y 68.5069,Z 192,A 26.7681,B 0.4923,C -0.0173,E1 0.6373,E2 428.1667} C_DIS
LIN {X 124.6395,Y 64.3972,Z 192,A 25.214,B 0.4923,C -0.0137,E1 0.6393,E2 429.6802} C_DIS
LIN {X 126.7993,Y 60.029,Z 192,A 23.7466,B 0.4925,C -0.0105,E1 0.641,E2 431.0865} C_DIS
LIN {X 128.6342,Y 55.9882,Z 192,A 22.4065,B 0.4925,C -0.0075,E1 0.6425,E2 432.3708} C_DIS
LIN {X 129.982,Y 52.7838,Z 192,A 21.1822,B 0.4925,C -0.0045,E1 0.6438,E2 433.572} C_DIS
LIN {X 131.2674,Y 49.5004,Z 192,A 20.0907,B 0.4925,C -0.002,E1 0.6448,E2 434.6219} C_DIS
LIN {X 132.4697,Y 46.1863,Z 192,A 18.9725,B 0.4925,C 0.0006,E1 0.6458,E2 435.7014} C_DIS
LIN {X 133.5071,Y 43.0974,Z 192,A 17.8739,B 0.4925,C 0.0032,E1 0.6468,E2 436.772} C_DIS
LIN {X 134.7017,Y 39.2028,Z 192,A 16.2103,B 0.4925,C 0.0078,E1 0.6481,E2 438.4363} C_DIS
LIN {X 135.8993,Y 34.8262,Z 192,A 15.1283,B 0.4925,C 0.0097,E1 0.6488,E2 439.4236} C_DIS
LIN {X 136.8777,Y 30.7591,Z 192,A 13.6394,B 0.4924,C 0.0135,E1 0.6497,E2 440.8859} C_DIS
LIN {X 138.1671,Y 24.3188,Z 192,A 11.5818,B 0.4922,C 0.0183,E1 0.6507,E2 442.8659} C_DIS
LIN {X 138.8502,Y 20.0522,Z 192,A 10.2421,B 0.4922,C 0.0214,E1 0.6513,E2 444.1522} C_DIS
LIN {X 139.4442,Y 15.3913,Z 192,A 8.8102,B 0.4919,C 0.0247,E1 0.6517,E2 445.5225} C_DIS
LIN {X 139.7956,Y 11.7737,Z 192,A 7.6613,B 0.4919,C 0.0274,E1 0.652,E2 446.6286} C_DIS
LIN {X 140.0685,Y 7.9228,Z 192,A 6.3561,B 0.4916,C 0.0306,E1 0.6522,E2 447.8993} C_DIS
LIN {X 140.2422,Y 3.6938,Z 192,A 5.0509,B 0.4914,C 0.0337,E1 0.6524,E2 449.1499} C_DIS
LIN {X 140.2931,Y -0.2142,Z 192,A 3.7312,B 0.4912,C 0.0369,E1 0.6524,E2 450.4342} C_DIS
LIN {X 140.2257,Y -4.2847,Z 192,A 2.4861,B 0.491,C 0.0398,E1 0.6524,E2 451.6247} C_DIS
LIN {X 140.04,Y -8.3853,Z 192,A 1.1943,B 0.4907,C 0.0428,E1 0.6521,E2 452.866} C_DIS
LIN {X 139.7482,Y -12.3356,Z 192,A -0.1254,B 0.4904,C 0.046,E1 0.6518,E2 454.1466} C_DIS
LIN {X 139.3202,Y -16.4724,Z 192,A -1.3726,B 0.4901,C 0.0488,E1 0.6515,E2 455.3337} C_DIS
LIN {X 138.8962,Y -19.7297,Z 192,A -2.4559,B 0.4899,C 0.0514,E1 0.6511,E2 456.3827} C_DIS
LIN {X 138.3693,Y -23.1375,Z 192,A -3.5664,B 0.4896,C 0.054,E1 0.6506,E2 457.4533} C_DIS
LIN {X 137.7109,Y -26.7824,Z 192,A -4.7639,B 0.4893,C 0.0568,E1 0.65,E2 458.6085} C_DIS
LIN {X 136.8903,Y -30.704,Z 192,A -5.9633,B 0.489,C 0.0595,E1 0.6493,E2 459.7487} C_DIS
LIN {X 136.3158,Y -33.1583,Z 192,A -6.8248,B 0.4887,C 0.0615,E1 0.6488,E2 460.5874} C_DIS
LIN {X 135.2641,Y -37.2201,Z 192,A -8.2507,B 0.4883,C 0.065,E1 0.6478,E2 461.9743} C_DIS
LIN {X 134.1922,Y -40.9125,Z 192,A -9.423,B 0.4879,C 0.0676,E1 0.6469,E2 463.0919} C_DIS
LIN {X 132.4258,Y -46.3129,Z 192,A -11.2782,B 0.4873,C 0.0718,E1 0.6453,E2 464.8832} C_DIS
LIN {X 130.9057,Y -50.4499,Z 192,A -12.7258,B 0.4868,C 0.0751,E1 0.6439,E2 466.282} C_DIS
LIN {X 129.5496,Y -53.8358,Z 192,A -13.8555,B 0.4864,C 0.0776,E1 0.6428,E2 467.3614} C_DIS
LIN {X 127.8426,Y -57.7742,Z 192,A -15.4782,B 0.4858,C 0.0817,E1 0.641,E2 468.9667} C_DIS
LIN {X 126.407,Y -60.85,Z 192,A -16.4464,B 0.4854,C 0.0835,E1 0.6399,E2 469.8758} C_DIS
LIN {X 124.4587,Y -64.7427,Z 192,A -17.8011,B 0.4849,C 0.0864,E1 0.6382,E2 471.1707} C_DIS
LIN {X 122.9443,Y -67.5779,Z 192,A -18.84,B 0.4845,C 0.0886,E1 0.6369,E2 472.1708} C_DIS
LIN {X 120.2012,Y -72.3437,Z 192,A -20.7985,B 0.4837,C 0.0932,E1 0.6341,E2 474.0891} C_DIS
LIN {X 118.5026,Y -75.0937,Z 192,A -21.7091,B 0.4834,C 0.0948,E1 0.6329,E2 474.9407} C_DIS
LIN {X 116.1163,Y -78.733,Z 192,A -23.1239,B 0.4828,C 0.0978,E1 0.6307,E2 476.3036} C_DIS
LIN {X 113.4854,Y -82.4801,Z 192,A -24.6406,B 0.4821,C 0.101,E1 0.6283,E2 477.7694} C_DIS
LIN {X 110.8264,Y -86.0197,Z 192,A -26.0904,B 0.4815,C 0.1039,E1 0.6259,E2 479.1674} C_DIS
LIN {X 107.939,Y -89.6163,Z 192,A -27.6153,B 0.4808,C 0.107,E1 0.6233,E2 480.6402} C_DIS
LIN {X 104.9339,Y -93.1172,Z 192,A -29.1195,B 0.4801,C 0.11,E1 0.6206,E2 482.0889} C_DIS
LIN {X 101.8445,Y -96.4866,Z 192,A -30.6095,B 0.4795,C 0.1128,E1 0.6178,E2 483.5237} C_DIS
LIN {X 98.8135,Y -99.588,Z 192,A -32.0433,B 0.4788,C 0.1156,E1 0.615,E2 484.9078} C_DIS
LIN {X 95.8777,Y -102.4181,Z 192,A -33.4621,B 0.4781,C 0.1184,E1 0.6122,E2 486.2906} C_DIS
LIN {X 92.4864,Y -105.4905,Z 192,A -34.9734,B 0.4774,C 0.1212,E1 0.6091,E2 487.749} C_DIS
LIN {X 89.0915,Y -108.3732,Z 192,A -36.4909,B 0.4767,C 0.124,E1 0.6059,E2 489.2219} C_DIS
LIN {X 85.7518,Y -111.034,Z 192,A -37.9116,B 0.4761,C 0.1265,E1 0.6028,E2 490.5944} C_DIS
LIN {X 82.0535,Y -113.7946,Z 192,A -39.4484,B 0.4753,C 0.1291,E1 0.5994,E2 492.0792} C_DIS
LIN {X 78.5896,Y -116.2134,Z 192,A -40.8474,B 0.4747,C 0.1315,E1 0.5962,E2 493.4291} C_DIS
LIN {X 75.0451,Y -118.5333,Z 192,A -42.3456,B 0.474,C 0.1341,E1 0.5927,E2 494.8929} C_DIS
LIN {X 71.2239,Y -120.868,Z 192,A -43.8557,B 0.4733,C 0.1365,E1 0.5891,E2 496.355} C_DIS
LIN {X 64.854,Y -124.4003,Z 192,A -46.3389,B 0.4721,C 0.1404,E1 0.583,E2 498.7639} C_DIS
LIN {X 62.3701,Y -125.6638,Z 192,A -48.0233,B 0.471,C 0.1443,E1 0.5784,E2 500.5345} C_DIS
LIN {X 55.9396,Y -128.6552,Z 192,A -49.7011,B 0.4707,C 0.1453,E1 0.5745,E2 502.024} C_DIS
LIN {X 52.7838,Y -129.982,Z 192,A -50.9231,B 0.4701,C 0.147,E1 0.5713,E2 503.2194} C_DIS
LIN {X 49.1833,Y -131.3862,Z 192,A -52.1707,B 0.4696,C 0.1486,E1 0.568,E2 504.416} C_DIS
LIN {X 46.401,Y -132.3953,Z 192,A -53.3044,B 0.4691,C 0.1503,E1 0.565,E2 505.5388} C_DIS
LIN {X 43.7104,Y -133.3085,Z 192,A -54.6376,B 0.4683,C 0.1526,E1 0.5612,E2 506.9003} C_DIS
LIN {X 39.8424,Y -134.5144,Z 192,A -55.76,B 0.4681,C 0.1535,E1 0.5583,E2 507.9397} C_DIS
LIN {X 36.2152,Y -135.5353,Z 192,A -57.0611,B 0.4676,C 0.155,E1 0.5548,E2 509.2042} C_DIS
LIN {X 33.312,Y -136.2787,Z 192,A -58.1826,B 0.4671,C 0.1564,E1 0.5517,E2 510.3104} C_DIS
LIN {X 27.8546,Y -137.4974,Z 192,A -60.3795,B 0.4661,C 0.1592,E1 0.5454,E2 512.4951} C_DIS
LIN {X 24.5506,Y -138.1256,Z 192,A -61.3115,B 0.466,C 0.1597,E1 0.543,E2 513.3577} C_DIS
LIN {X 21.424,Y -138.6449,Z 192,A -62.4829,B 0.4655,C 0.1609,E1 0.5396,E2 514.5104} C_DIS
LIN {X 18.0073,Y -139.1302,Z 192,A -63.7897,B 0.4651,C 0.1623,E1 0.5359,E2 515.8018} C_DIS
LIN {X 13.6687,Y -139.6233,Z 192,A -65.3821,B 0.4645,C 0.1638,E1 0.5314,E2 517.3649} C_DIS
LIN {X 9.9855,Y -139.9349,Z 192,A -66.7483,B 0.4641,C 0.165,E1 0.5274,E2 518.7092} C_DIS
LIN {X 5.6034,Y -140.1787,Z 192,A -68.3914,B 0.4636,C 0.1664,E1 0.5227,E2 520.3295} C_DIS
LIN {X 1.0037,Y -140.2868,Z 192,A -70.0429,B 0.4632,C 0.1675,E1 0.518,E2 521.9456} C_DIS
Enddeposition()
LIN {X 1.0037,Y -140.2868,Z 192,A -70.0429,B 0.4632,C 0.1675,E1 0.518,E2 521.9456} C_DIS
Startdeposition()
$VEL.CP = VEL_PRINT
LIN {X 1.8349,Y -141.1786,Z 192,A -70.9653,B 0.5372,C 0.1729,E1 0.5897,E2 523.0656} C_DIS
LIN {X 1.8349,Y -141.1786,Z 192,A -70.9671,B 0.5372,C 0.1729,E1 0.5897,E2 523.0677} C_DIS
LIN {X 6.0237,Y -141.062,Z 192,A -69.4763,B 0.5375,C 0.1719,E1 0.5939,E2 521.6095} C_DIS
LIN {X 10.1644,Y -140.8232,Z 192,A -67.9063,B 0.5379,C 0.1707,E1 0.5984,E2 520.0564} C_DIS
LIN {X 14.219,Y -140.4735,Z 192,A -66.2814,B 0.5384,C 0.1691,E1 0.6031,E2 518.4347} C_DIS
LIN {X 18.4595,Y -139.9775,Z 192,A -64.7633,B 0.5388,C 0.1679,E1 0.6073,E2 516.9497} C_DIS
LIN {X 23.0412,Y -139.2967,Z 192,A -63.1783,B 0.5392,C 0.1666,E1 0.6117,E2 515.4104} C_DIS
LIN {X 30.9612,Y -137.7536,Z 192,A -60.2737,B 0.5401,C 0.1637,E1 0.6198,E2 512.5624} C_DIS
LIN {X 35.148,Y -136.745,Z 192,A -58.4771,B 0.5409,C 0.1612,E1 0.6249,E2 510.7569} C_DIS
LIN {X 38.5259,Y -135.8323,Z 192,A -57.3436,B 0.5412,C 0.1601,E1 0.6279,E2 509.6678} C_DIS
LIN {X 44.3271,Y -134.0506,Z 192,A -55.1865,B 0.5419,C 0.1576,E1 0.6337,E2 507.5573} C_DIS
LIN {X 47.3522,Y -133.013,Z 192,A -53.9506,B 0.5424,C 0.1558,E1 0.637,E2 506.3302} C_DIS
LIN {X 51.2626,Y -131.5542,Z 192,A -52.559,B 0.5429,C 0.1541,E1 0.6406,E2 504.9849} C_DIS
LIN {X 54.0741,Y -130.4242,Z 192,A -51.4858,B 0.5433,C 0.1527,E1 0.6434,E2 503.9354} C_DIS
LIN {X 57.3131,Y -129.0336,Z 192,A -49.713,B 0.5443,C 0.1491,E1 0.6482,E2 502.1075} C_DIS
LIN {X 61.9041,Y -126.896,Z 192,A -48.3751,B 0.5446,C 0.1481,E1 0.6514,E2 500.8809} C_DIS
LIN {X 64.6338,Y -125.5278,Z 192,A -46.8577,B 0.5455,C 0.1449,E1 0.6553,E2 499.3188} C_DIS
LIN {X 69.1099,Y -123.1208,Z 192,A -45.4987,B 0.5458,C 0.1436,E1 0.6585,E2 498.0685} C_DIS
LIN {X 73.1826,Y -120.7445,Z 192,A -43.8874,B 0.5464,C 0.1411,E1 0.6623,E2 496.5028} C_DIS
LIN {X 76.9835,Y -118.3574,Z 192,A -42.3082,B 0.5471,C 0.1385,E1 0.666,E2 494.9597} C_DIS
LIN {X 80.7272,Y -115.8362,Z 192,A -40.7746,B 0.5478,C 0.136,E1 0.6695,E2 493.4709} C_DIS
LIN {X 84.2001,Y -113.337,Z 192,A -39.2697,B 0.5484,C 0.1333,E1 0.6729,E2 492.0003} C_DIS
LIN {X 87.7734,Y -110.5928,Z 192,A -37.7302,B 0.5491,C 0.1306,E1 0.6762,E2 490.5039} C_DIS
LIN {X 91.1433,Y -107.833,Z 192,A -36.2057,B 0.5497,C 0.1278,E1 0.6795,E2 489.0153} C_DIS
LIN {X 94.5844,Y -104.8277,Z 192,A -34.6535,B 0.5504,C 0.1249,E1 0.6827,E2 487.5079} C_DIS
LIN {X 97.986,Y -101.655,Z 192,A -33.0972,B 0.551,C 0.1221,E1 0.6858,E2 486.0006} C_DIS
LIN {X 101.0434,Y -98.6167,Z 192,A -31.6497,B 0.5516,C 0.1193,E1 0.6886,E2 484.5976} C_DIS
LIN {X 104.1197,Y -95.3628,Z 192,A -30.1598,B 0.5522,C 0.1165,E1 0.6913,E2 483.1559} C_DIS
LIN {X 106.9477,Y -92.1796,Z 192,A -28.7003,B 0.5528,C 0.1136,E1 0.694,E2 481.7354} C_DIS
LIN {X 109.9124,Y -88.6237,Z 192,A -27.1709,B 0.5534,C 0.1105,E1 0.6966,E2 480.2572} C_DIS
LIN {X 112.491,Y -85.3277,Z 192,A -25.7178,B 0.554,C 0.1075,E1 0.6991,E2 478.8395} C_DIS
LIN {X 115.1618,Y -81.6872,Z 192,A -24.197,B 0.5546,C 0.1043,E1 0.7015,E2 477.3637} C_DIS
LIN {X 117.6508,Y -78.06,Z 192,A -22.7612,B 0.5552,C 0.1014,E1 0.7037,E2 475.9786} C_DIS
LIN {X 119.5154,Y -75.1733,Z 192,A -21.1232,B 0.556,C 0.0968,E1 0.7062,E2 474.3033} C_DIS
LIN {X 122.4833,Y -70.2342,Z 192,A -19.9241,B 0.5562,C 0.0958,E1 0.7077,E2 473.2708} C_DIS
LIN {X 124.4337,Y -66.7172,Z 192,A -18.2983,B 0.5569,C 0.0917,E1 0.7098,E2 471.6448} C_DIS
LIN {X 126.2584,Y -63.1966,Z 192,A -16.6543,B 0.5576,C 0.0873,E1 0.7119,E2 469.9945} C_DIS
LIN {X 128.442,Y -58.6299,Z 192,A -15.4529,B 0.5578,C 0.0857,E1 0.7132,E2 468.916} C_DIS
LIN {X 130.0778,Y -54.9035,Z 192,A -14.0584,B 0.5583,C 0.0825,E1 0.7147,E2 467.5574} C_DIS
LIN {X 131.423,Y -51.6003,Z 192,A -13.0251,B 0.5586,C 0.0805,E1 0.7157,E2 466.5827} C_DIS
LIN {X 132.7022,Y -48.2142,Z 192,A -11.7535,B 0.559,C 0.0774,E1 0.7169,E2 465.3384} C_DIS
LIN {X 133.6198,Y -45.6133,Z 192,A -10.7862,B 0.5594,C 0.0751,E1 0.7178,E2 464.3921} C_DIS
LIN {X 135.2935,Y -40.3805,Z 192,A -8.958,B 0.5599,C 0.0708,E1 0.7193,E2 462.6195} C_DIS
LIN {X 136.1428,Y -37.4157,Z 192,A -7.9926,B 0.5602,C 0.0687,E1 0.7199,E2 461.6938} C_DIS
LIN {X 136.9837,Y -34.2077,Z 192,A -6.9513,B 0.5605,C 0.0664,E1 0.7206,E2 460.6945} C_DIS
LIN {X 137.8816,Y -30.3884,Z 192,A -5.563,B 0.5609,C 0.0629,E1 0.7215,E2 459.3338} C_DIS
Enddeposition()
END
